TEXTLIST S6_Alarms
  0 = 'Station 6 Clamp A1 Failed to Advance... Check Q1.0...' | German: 'S6 0 Row 1 Failed To Advance.. Check Qxxx.x German' | French: 'S6 0 Row 1 Failed To Advance.. Check Qxxx.x French' | 汉语: '汉语'
  1 = 'Station 6 Clamp A1 Failed to Return... Check Q1.1...' | German: 'S6 1 Row 1 Failed To Return.. Check Qxxx.x German' | French: 'S6 1 Row 1 Failed To Return.. Check Qxxx.x French' | 汉语: '汉语'
  2 = 'Station 6 Clamp A1 Lost Advanced... Check I1.0...' | German: 'S6 2 Row 1 Lost Advance Position... Check Ixxx.x German' | French: 'S6 2 Row 1 Lost Advance Position... Check Ixxx.x French' | 汉语: '汉语'
  3 = 'Station 6 Clamp A1 Lost Returned... Check I1.1...' | German: 'S6 3 Row 1 Lost Return Position... Check Ixxx.x German' | French: 'S6 3 Row 1 Lost Return Position... Check Ixxx.x French' | 汉语: '汉语'
  4 = 'Station 6 Clamp A1 Switch Fault... Check I1.0, I1.1...' | German: 'S6 4 Row 1 Switch Fault... Check Ixxx.x / Ixxx.x German' | French: 'S6 4 Row 1 Switch Fault... Check Ixxx.x / Ixxx.x French'
  5 = 'Spare' | German: 'S6 5 Row 1 Spare Message German' | French: 'S6 5 Row 1 Spare Message French'
  6 = 'Spare' | German: 'S6 6 Row 1 Spare Message German' | French: 'S6 6 Row 1 Spare Message French'
  7 = 'Spare' | German: 'S6 7 Row 1 Spare Message German' | French: 'S6 7 Row 1 Spare Message French'
  8 = 'Spare' | German: 'S6 8 Row 1 Spare Message German' | French: 'S6 8 Row 1 Spare Message French'
  9 = 'Spare' | German: 'S6 9 Row 1 Spare Message German' | French: 'S6 9 Row 1 Spare Message French'
  10 = 'Lock Cylinder A2 Failed to Lock... Check Q1.2...' | German: 'S6 10 Row 2 Failed To Advance.. Check Qxxx.x German' | French: 'S6 10 Row 2 Failed To Advance.. Check Qxxx.x French'
  11 = 'Lock Cylinder A2 Failed to Unlock... Check Q1.3...' | German: 'S6 11 Row 2 Failed To Return.. Check Qxxx.x German' | French: 'S6 11 Row 2 Failed To Return.. Check Qxxx.x French'
  12 = 'Lock Cylinder A2 Lost Locked... Check I1.2...' | German: 'S6 12 Row 2 Lost Advance Position... Check Ixxx.x German' | French: 'S6 12 Row 2 Lost Advance Position... Check Ixxx.x French'
  13 = 'Lock Cylinder A2 Lost Unlocked... Check I1.3...' | German: 'S6 13 Row 2 Lost Return Position... Check Ixxx.x German' | French: 'S6 13 Row 2 Lost Return Position... Check Ixxx.x French'
  14 = 'Lock Cylinder A2 Switch Fault... Check I1.2, I1.3...' | German: 'S6 14 Row 2 Switch Fault... Check Ixxx.x / Ixxx.x German' | French: 'S6 14 Row 2 Switch Fault... Check Ixxx.x / Ixxx.x French'
  15 = 'Spare' | German: 'S6 15 Row 2 Spare Message German' | French: 'S6 15 Row 2 Spare Message French'
  16 = 'Spare' | German: 'S6 16 Row 2 Spare Message German' | French: 'S6 16 Row 2 Spare Message French'
  17 = 'Spare' | German: 'S6 17 Row 2 Spare Message German' | French: 'S6 17 Row 2 Spare Message French'
  18 = 'Spare' | German: 'S6 18 Row 2 Spare Message German' | French: 'S6 18 Row 2 Spare Message French'
  19 = 'Spare' | German: 'S6 19 Row 2 Spare Message German' | French: 'S6 19 Row 2 Spare Message French'
  20 = 'Urger Cylinder A3 Failed to Urge... Check Q1.4...' | German: 'S6 20 Row 3 Failed To Advance.. Check Qxxx.x German' | French: 'S6 20 Row 3 Failed To Advance.. Check Qxxx.x French'
  21 = 'Urger Cylinder A3 Failed to Return... Check Q1.5...' | German: 'S6 21 Row 3 Failed To Return.. Check Qxxx.x German' | French: 'S6 21 Row 3 Failed To Return.. Check Qxxx.x French'
  22 = 'Urger Cylinder A3 Lost Urged... Check I1.4...' | German: 'S6 22 Row 3 Lost Advance Position... Check Ixxx.x German' | French: 'S6 22 Row 3 Lost Advance Position... Check Ixxx.x French'
  23 = 'Urger Cylinder A3 Lost Returned... Check I1.5...' | German: 'S6 23 Row 3 Lost Return Position... Check Ixxx.x German' | French: 'S6 23 Row 3 Lost Return Position... Check Ixxx.x French'
  24 = 'Urger Cylinder A3 Switch Fault... Check I1.4, I1.5...' | German: 'S6 24 Row 3 Switch Fault... Check Ixxx.x / Ixxx.x German' | French: 'S6 24 Row 3 Switch Fault... Check Ixxx.x / Ixxx.x French'
  25 = 'Spare' | German: 'S6 25 Row 3 Spare Message German' | French: 'S6 25 Row 3 Spare Message French'
  26 = 'Spare' | German: 'S6 26 Row 3 Spare Message German' | French: 'S6 26 Row 3 Spare Message French'
  27 = 'Spare' | German: 'S6 27 Row 3 Spare Message German' | French: 'S6 27 Row 3 Spare Message French'
  28 = 'Spare' | German: 'S6 28 Row 3 Spare Message German' | French: 'S6 28 Row 3 Spare Message French'
  29 = 'Spare' | German: 'S6 29 Row 3 Spare Message German' | French: 'S6 29 Row 3 Spare Message French'
  30 = 'Clamp Cylinder A1 Failed to Advance... Check Q1.0...' | German: 'S6 30 Row 4 Failed To Advance.. Check Qxxx.x German' | French: 'S6 30 Row 4 Failed To Advance.. Check Qxxx.x French'
  31 = 'Clamp Cylinder A1 Failed to Return... Check Q1.1...' | German: 'S6 31 Row 4 Failed To Return.. Check Qxxx.x German' | French: 'S6 31 Row 4 Failed To Return.. Check Qxxx.x French'
  32 = 'Clamp Cylinder A1 Lost Advanced... Check I1.0...' | German: 'S6 32 Row 4 Lost Advance Position... Check Ixxx.x German' | French: 'S6 32 Row 4 Lost Advance Position... Check Ixxx.x French'
  33 = 'Clamp Cylinder A1 Lost Returned... Check I1.1...' | German: 'S6 33 Row 4 Lost Return Position... Check Ixxx.x German' | French: 'S6 33 Row 4 Lost Return Position... Check Ixxx.x French'
  34 = 'Clamp Cylinder A1 Switch Fault... Check I1.0, I1.1...' | German: 'S6 34 Row 4 Switch Fault... Check Ixxx.x / Ixxx.x German' | French: 'S6 34 Row 4 Switch Fault... Check Ixxx.x / Ixxx.x French'
  35 = 'Spare' | German: 'S6 35 Row 4 Spare Message German' | French: 'S6 35 Row 4 Spare Message French'
  36 = 'Spare' | German: 'S6 36 Row 4 Spare Message German' | French: 'S6 36 Row 4 Spare Message French'
  37 = 'Spare' | German: 'S6 37 Row 4 Spare Message German' | French: 'S6 37 Row 4 Spare Message French'
  38 = 'Spare' | German: 'S6 38 Row 4 Spare Message German' | French: 'S6 38 Row 4 Spare Message French'
  39 = 'Spare' | German: 'S6 39 Row 4 Spare Message German' | French: 'S6 39 Row 4 Spare Message French'
  40 = 'Clamp Cylinder A1 Failed to Advance... Check Q1.0...' | German: 'S6 40 Row 5 Failed To Advance.. Check Qxxx.x German' | French: 'S6 40 Row 5 Failed To Advance.. Check Qxxx.x French'
  41 = 'Clamp Cylinder A1 Failed to Return... Check Q1.1...' | German: 'S6 41 Row 5 Failed To Return.. Check Qxxx.x German' | French: 'S6 41 Row 5 Failed To Return.. Check Qxxx.x French'
  42 = 'Clamp Cylinder A1 Lost Advanced... Check I1.0...' | German: 'S6 42 Row 5 Lost Advance Position... Check Ixxx.x German' | French: 'S6 42 Row 5 Lost Advance Position... Check Ixxx.x French'
  43 = 'Clamp Cylinder A1 Lost Returned... Check I1.1...' | German: 'S6 43 Row 5 Lost Return Position... Check Ixxx.x German' | French: 'S6 43 Row 5 Lost Return Position... Check Ixxx.x French'
  44 = 'Clamp Cylinder A1 Switch Fault... Check I1.0, I1.1...' | German: 'S6 44 Row 5 Switch Fault... Check Ixxx.x / Ixxx.x German' | French: 'S6 44 Row 5 Switch Fault... Check Ixxx.x / Ixxx.x French'
  45 = 'Spare' | German: 'S6 45 Row 5 Spare Message German' | French: 'S6 45 Row 5 Spare Message French'
  46 = 'Spare' | German: 'S6 46 Row 5 Spare Message German' | French: 'S6 46 Row 5 Spare Message French'
  47 = 'Spare' | German: 'S6 47 Row 5 Spare Message German' | French: 'S6 47 Row 5 Spare Message French'
  48 = 'Spare' | German: 'S6 48 Row 5 Spare Message German' | French: 'S6 48 Row 5 Spare Message French'
  49 = 'Spare' | German: 'S6 49 Row 5 Spare Message German' | French: 'S6 49 Row 5 Spare Message French'
  50 = 'Clamp Cylinder A1 Failed to Advance... Check Q1.0...' | German: 'S6 50 Row 6 Failed To Advance.. Check Qxxx.x German' | French: 'S6 50 Row 6 Failed To Advance.. Check Qxxx.x French'
  51 = 'Clamp Cylinder A1 Failed to Return... Check Q1.1...' | German: 'S6 51 Row 6 Failed To Return.. Check Qxxx.x German' | French: 'S6 51 Row 6 Failed To Return.. Check Qxxx.x French'
  52 = 'Clamp Cylinder A1 Lost Advanced... Check I1.0...' | German: 'S6 52 Row 6 Lost Advance Position... Check Ixxx.x German' | French: 'S6 52 Row 6 Lost Advance Position... Check Ixxx.x French'
  53 = 'Clamp Cylinder A1 Lost Returned... Check I1.1...' | German: 'S6 53 Row 6 Lost Return Position... Check Ixxx.x German' | French: 'S6 53 Row 6 Lost Return Position... Check Ixxx.x French'
  54 = 'Clamp Cylinder A1 Switch Fault... Check I1.0, I1.1...' | German: 'S6 54 Row 6 Switch Fault... Check Ixxx.x / Ixxx.x German' | French: 'S6 54 Row 6 Switch Fault... Check Ixxx.x / Ixxx.x French'
  55 = 'Spare' | German: 'S6 55 Row 6 Spare Message German' | French: 'S6 55 Row 6 Spare Message French'
  56 = 'Spare' | German: 'S6 56 Row 6 Spare Message German' | French: 'S6 56 Row 6 Spare Message French'
  57 = 'Spare' | German: 'S6 57 Row 6 Spare Message German' | French: 'S6 57 Row 6 Spare Message French'
  58 = 'Spare' | German: 'S6 58 Row 6 Spare Message German' | French: 'S6 58 Row 6 Spare Message French'
  59 = 'Spare' | German: 'S6 59 Row 6 Spare Message German' | French: 'S6 59 Row 6 Spare Message French'
  60 = 'Clamp Cylinder A1 Failed to Advance... Check Q1.0...' | German: 'S6 60 Row 7 Failed To Advance.. Check Qxxx.x German' | French: 'S6 60 Row 7 Failed To Advance.. Check Qxxx.x French'
  61 = 'Clamp Cylinder A1 Failed to Return... Check Q1.1...' | German: 'S6 61 Row 7 Failed To Return.. Check Qxxx.x German' | French: 'S6 61 Row 7 Failed To Return.. Check Qxxx.x French'
  62 = 'Clamp Cylinder A1 Lost Advanced... Check I1.0...' | German: 'S6 62 Row 7 Lost Advance Position... Check Ixxx.x German' | French: 'S6 62 Row 7 Lost Advance Position... Check Ixxx.x French'
  63 = 'Clamp Cylinder A1 Lost Returned... Check I1.1...' | German: 'S6 63 Row 7 Lost Return Position... Check Ixxx.x German' | French: 'S6 63 Row 7 Lost Return Position... Check Ixxx.x French'
  64 = 'Clamp Cylinder A1 Switch Fault... Check I1.0, I1.1...' | German: 'S6 64 Row 7 Switch Fault... Check Ixxx.x / Ixxx.x German' | French: 'S6 64 Row 7 Switch Fault... Check Ixxx.x / Ixxx.x French'
  65 = 'Spare' | German: 'S6 65 Row 7 Spare Message German' | French: 'S6 65 Row 7 Spare Message French'
  66 = 'Spare' | German: 'S6 66 Row 7 Spare Message German' | French: 'S6 66 Row 7 Spare Message French'
  67 = 'Spare' | German: 'S6 67 Row 7 Spare Message German' | French: 'S6 67 Row 7 Spare Message French'
  68 = 'Spare' | German: 'S6 68 Row 7 Spare Message German' | French: 'S6 68 Row 7 Spare Message French'
  69 = 'Spare' | German: 'S6 69 Row 7 Spare Message German' | French: 'S6 69 Row 7 Spare Message French'
  70 = 'Clamp Cylinder A1 Failed to Advance... Check Q1.0...' | German: 'S6 70 Row 8 Failed To Advance.. Check Qxxx.x German' | French: 'S6 70 Row 8 Failed To Advance.. Check Qxxx.x French'
  71 = 'Clamp Cylinder A1 Failed to Return... Check Q1.1...' | German: 'S6 71 Row 8 Failed To Return.. Check Qxxx.x German' | French: 'S6 71 Row 8 Failed To Return.. Check Qxxx.x French'
  72 = 'Clamp Cylinder A1 Lost Advanced... Check I1.0...' | German: 'S6 72 Row 8 Lost Advance Position... Check Ixxx.x German' | French: 'S6 72 Row 8 Lost Advance Position... Check Ixxx.x French'
  73 = 'Clamp Cylinder A1 Lost Returned... Check I1.1...' | German: 'S6 73 Row 8 Lost Return Position... Check Ixxx.x German' | French: 'S6 73 Row 8 Lost Return Position... Check Ixxx.x French'
  74 = 'Clamp Cylinder A1 Switch Fault... Check I1.0, I1.1...' | German: 'S6 74 Row 8 Switch Fault... Check Ixxx.x / Ixxx.x German' | French: 'S6 74 Row 8 Switch Fault... Check Ixxx.x / Ixxx.x French'
  75 = 'Spare' | German: 'S6 75 Row 8 Spare Message German' | French: 'S6 75 Row 8 Spare Message French'
  76 = 'Spare' | German: 'S6 76 Row 8 Spare Message German' | French: 'S6 76 Row 8 Spare Message French'
  77 = 'Spare' | German: 'S6 77 Row 8 Spare Message German' | French: 'S6 77 Row 8 Spare Message French'
  78 = 'Spare' | German: 'S6 78 Row 8 Spare Message German' | French: 'S6 78 Row 8 Spare Message French'
  79 = 'Spare' | German: 'S6 79 Row 8 Spare Message German' | French: 'S6 79 Row 8 Spare Message French'
  80 = 'Clamp Cylinder A1 Failed to Advance... Check Q1.0...' | German: 'S6 80 Row 9 Failed To Advance.. Check Qxxx.x German' | French: 'S6 80 Row 9 Failed To Advance.. Check Qxxx.x French'
  81 = 'Clamp Cylinder A1 Failed to Return... Check Q1.1...' | German: 'S6 81 Row 9 Failed To Return.. Check Qxxx.x German' | French: 'S6 81 Row 9 Failed To Return.. Check Qxxx.x French'
  82 = 'Clamp Cylinder A1 Lost Advanced... Check I1.0...' | German: 'S6 82 Row 9 Lost Advance Position... Check Ixxx.x German' | French: 'S6 82 Row 9 Lost Advance Position... Check Ixxx.x French'
  83 = 'Clamp Cylinder A1 Lost Returned... Check I1.1...' | German: 'S6 83 Row 9 Lost Return Position... Check Ixxx.x German' | French: 'S6 83 Row 9 Lost Return Position... Check Ixxx.x French'
  84 = 'Clamp Cylinder A1 Switch Fault... Check I1.0, I1.1...' | German: 'S6 84 Row 9 Switch Fault... Check Ixxx.x / Ixxx.x German' | French: 'S6 84 Row 9 Switch Fault... Check Ixxx.x / Ixxx.x French'
  85 = 'Spare' | German: 'S6 85 Row 9 Spare Message German' | French: 'S6 85 Row 9 Spare Message French'
  86 = 'Spare' | German: 'S6 86 Row 9 Spare Message German' | French: 'S6 86 Row 9 Spare Message French'
  87 = 'Spare' | German: 'S6 87 Row 9 Spare Message German' | French: 'S6 87 Row 9 Spare Message French'
  88 = 'Spare' | German: 'S6 88 Row 9 Spare Message German' | French: 'S6 88 Row 9 Spare Message French'
  89 = 'Spare' | German: 'S6 89 Row 9 Spare Message German' | French: 'S6 89 Row 9 Spare Message French'
  90 = 'Clamp Cylinder A1 Failed to Advance... Check Q1.0...' | German: 'S6 90 Row 10 Failed To Advance.. Check Qxxx.x German' | French: 'S6 90 Row 10 Failed To Advance.. Check Qxxx.x French'
  91 = 'Clamp Cylinder A1 Failed to Return... Check Q1.1...' | German: 'S6 91 Row 10 Failed To Return.. Check Qxxx.x German' | French: 'S6 91 Row 10 Failed To Return.. Check Qxxx.x French'
  92 = 'Clamp Cylinder A1 Lost Advanced... Check I1.0...' | German: 'S6 92 Row 10 Lost Advance Position... Check Ixxx.x German' | French: 'S6 92 Row 10 Lost Advance Position... Check Ixxx.x French'
  93 = 'Clamp Cylinder A1 Lost Returned... Check I1.1...' | German: 'S6 93 Row 10 Lost Return Position... Check Ixxx.x German' | French: 'S6 93 Row 10 Lost Return Position... Check Ixxx.x French'
  94 = 'Clamp Cylinder A1 Switch Fault... Check I1.0, I1.1...' | German: 'S6 94 Row 10 Switch Fault... Check Ixxx.x / Ixxx.x German' | French: 'S6 94 Row 10 Switch Fault... Check Ixxx.x / Ixxx.x French'
  95 = 'Spare' | German: 'S6 95 Row 10 Spare Message German' | French: 'S6 95 Row 10 Spare Message French'
  96 = 'Spare' | German: 'S6 96 Row 10 Spare Message German' | French: 'S6 96 Row 10 Spare Message French'
  97 = 'Spare' | German: 'S6 97 Row 10 Spare Message German' | French: 'S6 97 Row 10 Spare Message French'
  98 = 'Spare' | German: 'S6 98 Row 10 Spare Message German' | French: 'S6 98 Row 10 Spare Message French'
  99 = 'Spare' | German: 'S6 99 Row 10 Spare Message German' | French: 'S6 99 Row 10 Spare Message French'
  100 = 'Clamp Cylinder A1 Failed to Advance... Check Q1.0...' | German: 'S6 100 Row 11 Failed To Advance.. Check Qxxx.x German' | French: 'S6 100 Row 11 Failed To Advance.. Check Qxxx.x French'
  101 = 'Clamp Cylinder A1 Failed to Return... Check Q1.1...' | German: 'S6 101 Row 11 Failed To Return.. Check Qxxx.x German' | French: 'S6 101 Row 11 Failed To Return.. Check Qxxx.x French'
  102 = 'Clamp Cylinder A1 Lost Advanced... Check I1.0...' | German: 'S6 102 Row 11 Lost Advance Position... Check Ixxx.x German' | French: 'S6 102 Row 11 Lost Advance Position... Check Ixxx.x French'
  103 = 'Clamp Cylinder A1 Lost Returned... Check I1.1...' | German: 'S6 103 Row 11 Lost Return Position... Check Ixxx.x German' | French: 'S6 103 Row 11 Lost Return Position... Check Ixxx.x French'
  104 = 'Clamp Cylinder A1 Switch Fault... Check I1.0, I1.1...' | German: 'S6 104 Row 11 Switch Fault... Check Ixxx.x / Ixxx.x German' | French: 'S6 104 Row 11 Switch Fault... Check Ixxx.x / Ixxx.x French'
  105 = 'Spare' | German: 'S6 105 Row 11 Spare Message German' | French: 'S6 105 Row 11 Spare Message French'
  106 = 'Spare' | German: 'S6 106 Row 11 Spare Message German' | French: 'S6 106 Row 11 Spare Message French'
  107 = 'Spare' | German: 'S6 107 Row 11 Spare Message German' | French: 'S6 107 Row 11 Spare Message French'
  108 = 'Spare' | German: 'S6 108 Row 11 Spare Message German' | French: 'S6 108 Row 11 Spare Message French'
  109 = 'Spare' | German: 'S6 109 Row 11 Spare Message German' | French: 'S6 109 Row 11 Spare Message French'
  110 = 'Clamp Cylinder A1 Failed to Advance... Check Q1.0...' | German: 'S6 110 Row 12 Failed To Advance.. Check Qxxx.x German' | French: 'S6 110 Row 12 Failed To Advance.. Check Qxxx.x French'
  111 = 'Clamp Cylinder A1 Failed to Return... Check Q1.1...' | German: 'S6 111 Row 12 Failed To Return.. Check Qxxx.x German' | French: 'S6 111 Row 12 Failed To Return.. Check Qxxx.x French'
  112 = 'Clamp Cylinder A1 Lost Advanced... Check I1.0...' | German: 'S6 112 Row 12 Lost Advance Position... Check Ixxx.x German' | French: 'S6 112 Row 12 Lost Advance Position... Check Ixxx.x French'
  113 = 'Clamp Cylinder A1 Lost Returned... Check I1.1...' | German: 'S6 113 Row 12 Lost Return Position... Check Ixxx.x German' | French: 'S6 113 Row 12 Lost Return Position... Check Ixxx.x French'
  114 = 'Clamp Cylinder A1 Switch Fault... Check I1.0, I1.1...' | German: 'S6 114 Row 12 Switch Fault... Check Ixxx.x / Ixxx.x German' | French: 'S6 114 Row 12 Switch Fault... Check Ixxx.x / Ixxx.x French'
  115 = 'Spare' | German: 'S6 115 Row 12 Spare Message German' | French: 'S6 115 Row 12 Spare Message French'
  116 = 'Spare' | German: 'S6 116 Row 12 Spare Message German' | French: 'S6 116 Row 12 Spare Message French'
  117 = 'Spare' | German: 'S6 117 Row 12 Spare Message German' | French: 'S6 117 Row 12 Spare Message French'
  118 = 'Spare' | German: 'S6 118 Row 12 Spare Message German' | French: 'S6 118 Row 12 Spare Message French'
  119 = 'Spare' | German: 'S6 119 Row 12 Spare Message German' | French: 'S6 119 Row 12 Spare Message French'
  120 = 'Clamp Cylinder A1 Failed to Advance... Check Q1.0...' | German: 'S6 120 Row 13 Failed To Advance.. Check Qxxx.x German' | French: 'S6 120 Row 13 Failed To Advance.. Check Qxxx.x French'
  121 = 'Clamp Cylinder A1 Failed to Return... Check Q1.1...' | German: 'S6 121 Row 13 Failed To Return.. Check Qxxx.x German' | French: 'S6 121 Row 13 Failed To Return.. Check Qxxx.x French'
  122 = 'Clamp Cylinder A1 Lost Advanced... Check I1.0...' | German: 'S6 122 Row 13 Lost Advance Position... Check Ixxx.x German' | French: 'S6 122 Row 13 Lost Advance Position... Check Ixxx.x French'
  123 = 'Clamp Cylinder A1 Lost Returned... Check I1.1...' | German: 'S6 123 Row 13 Lost Return Position... Check Ixxx.x German' | French: 'S6 123 Row 13 Lost Return Position... Check Ixxx.x French'
  124 = 'Clamp Cylinder A1 Switch Fault... Check I1.0, I1.1...' | German: 'S6 124 Row 13 Switch Fault... Check Ixxx.x / Ixxx.x German' | French: 'S6 124 Row 13 Switch Fault... Check Ixxx.x / Ixxx.x French'
  125 = 'Spare' | German: 'S6 125 Row 13 Spare Message German' | French: 'S6 125 Row 13 Spare Message French'
  126 = 'Spare' | German: 'S6 126 Row 13 Spare Message German' | French: 'S6 126 Row 13 Spare Message French'
  127 = 'Spare' | German: 'S6 127 Row 13 Spare Message German' | French: 'S6 127 Row 13 Spare Message French'
  128 = 'Spare' | German: 'S6 128 Row 13 Spare Message German' | French: 'S6 128 Row 13 Spare Message French'
  129 = 'Spare' | German: 'S6 129 Row 13 Spare Message German' | French: 'S6 129 Row 13 Spare Message French'
  130 = 'Clamp Cylinder A1 Failed to Advance... Check Q1.0...' | German: 'S6 130 Row 14 Failed To Advance.. Check Qxxx.x German' | French: 'S6 130 Row 14 Failed To Advance.. Check Qxxx.x French'
  131 = 'Clamp Cylinder A1 Failed to Return... Check Q1.1...' | German: 'S6 131 Row 14 Failed To Return.. Check Qxxx.x German' | French: 'S6 131 Row 14 Failed To Return.. Check Qxxx.x French'
  132 = 'Clamp Cylinder A1 Lost Advanced... Check I1.0...' | German: 'S6 132 Row 14 Lost Advance Position... Check Ixxx.x German' | French: 'S6 132 Row 14 Lost Advance Position... Check Ixxx.x French'
  133 = 'Clamp Cylinder A1 Lost Returned... Check I1.1...' | German: 'S6 133 Row 14 Lost Return Position... Check Ixxx.x German' | French: 'S6 133 Row 14 Lost Return Position... Check Ixxx.x French'
  134 = 'Clamp Cylinder A1 Switch Fault... Check I1.0, I1.1...' | German: 'S6 134 Row 14 Switch Fault... Check Ixxx.x / Ixxx.x German' | French: 'S6 134 Row 14 Switch Fault... Check Ixxx.x / Ixxx.x French'
  135 = 'Spare' | German: 'S6 135 Row 14 Spare Message German' | French: 'S6 135 Row 14 Spare Message French'
  136 = 'Spare' | German: 'S6 136 Row 14 Spare Message German' | French: 'S6 136 Row 14 Spare Message French'
  137 = 'Spare' | German: 'S6 137 Row 14 Spare Message German' | French: 'S6 137 Row 14 Spare Message French'
  138 = 'Spare' | German: 'S6 138 Row 14 Spare Message German' | French: 'S6 138 Row 14 Spare Message French'
  139 = 'Spare' | German: 'S6 139 Row 14 Spare Message German' | French: 'S6 139 Row 14 Spare Message French'
  140 = 'Clamp Cylinder A1 Failed to Advance... Check Q1.0...' | German: 'S6 140 Row 15 Failed To Advance.. Check Qxxx.x German' | French: 'S6 140 Row 15 Failed To Advance.. Check Qxxx.x French'
  141 = 'Clamp Cylinder A1 Failed to Return... Check Q1.1...' | German: 'S6 141 Row 15 Failed To Return.. Check Qxxx.x German' | French: 'S6 141 Row 15 Failed To Return.. Check Qxxx.x French'
  142 = 'Clamp Cylinder A1 Lost Advanced... Check I1.0...' | German: 'S6 142 Row 15 Lost Advance Position... Check Ixxx.x German' | French: 'S6 142 Row 15 Lost Advance Position... Check Ixxx.x French'
  143 = 'Clamp Cylinder A1 Lost Returned... Check I1.1...' | German: 'S6 143 Row 15 Lost Return Position... Check Ixxx.x German' | French: 'S6 143 Row 15 Lost Return Position... Check Ixxx.x French'
  144 = 'Clamp Cylinder A1 Switch Fault... Check I1.0, I1.1...' | German: 'S6 144 Row 15 Switch Fault... Check Ixxx.x / Ixxx.x German' | French: 'S6 144 Row 15 Switch Fault... Check Ixxx.x / Ixxx.x French'
  145 = 'Spare' | German: 'S6 145 Row 15 Spare Message German' | French: 'S6 145 Row 15 Spare Message French'
  146 = 'Spare' | German: 'S6 146 Row 15 Spare Message German' | French: 'S6 146 Row 15 Spare Message French'
  147 = 'Spare' | German: 'S6 147 Row 15 Spare Message German' | French: 'S6 147 Row 15 Spare Message French'
  148 = 'Spare' | German: 'S6 148 Row 15 Spare Message German' | French: 'S6 148 Row 15 Spare Message French'
  149 = 'Spare' | German: 'S6 149 Row 15 Spare Message German' | French: 'S6 149 Row 15 Spare Message French'
  150 = 'Clamp Cylinder A1 Failed to Advance... Check Q1.0...' | German: 'S6 150 Row 16 Failed To Advance.. Check Qxxx.x German' | French: 'S6 150 Row 16 Failed To Advance.. Check Qxxx.x French'
  151 = 'Clamp Cylinder A1 Failed to Return... Check Q1.1...' | German: 'S6 151 Row 16 Failed To Return.. Check Qxxx.x German' | French: 'S6 151 Row 16 Failed To Return.. Check Qxxx.x French'
  152 = 'Clamp Cylinder A1 Lost Advanced... Check I1.0...' | German: 'S6 152 Row 16 Lost Advance Position... Check Ixxx.x German' | French: 'S6 152 Row 16 Lost Advance Position... Check Ixxx.x French'
  153 = 'Clamp Cylinder A1 Lost Returned... Check I1.1...' | German: 'S6 153 Row 16 Lost Return Position... Check Ixxx.x German' | French: 'S6 153 Row 16 Lost Return Position... Check Ixxx.x French'
  154 = 'Clamp Cylinder A1 Switch Fault... Check I1.0, I1.1...' | German: 'S6 154 Row 16 Switch Fault... Check Ixxx.x / Ixxx.x German' | French: 'S6 154 Row 16 Switch Fault... Check Ixxx.x / Ixxx.x French'
  155 = 'Spare' | German: 'S6 155 Row 16 Spare Message German' | French: 'S6 155 Row 16 Spare Message French'
  156 = 'Spare' | German: 'S6 156 Row 16 Spare Message German' | French: 'S6 156 Row 16 Spare Message French'
  157 = 'Spare' | German: 'S6 157 Row 16 Spare Message German' | French: 'S6 157 Row 16 Spare Message French'
  158 = 'Spare' | German: 'S6 158 Row 16 Spare Message German' | French: 'S6 158 Row 16 Spare Message French'
  159 = 'Spare' | German: 'S6 159 Row 16 Spare Message German' | French: 'S6 159 Row 16 Spare Message French'
  160 = 'Clamp Cylinder A1 Failed to Advance... Check Q1.0...' | German: 'S6 160 Row 17 Failed To Advance.. Check Qxxx.x German' | French: 'S6 160 Row 17 Failed To Advance.. Check Qxxx.x French'
  161 = 'Clamp Cylinder A1 Failed to Return... Check Q1.1...' | German: 'S6 161 Row 17 Failed To Return.. Check Qxxx.x German' | French: 'S6 161 Row 17 Failed To Return.. Check Qxxx.x French'
  162 = 'Clamp Cylinder A1 Lost Advanced... Check I1.0...' | German: 'S6 162 Row 17 Lost Advance Position... Check Ixxx.x German' | French: 'S6 162 Row 17 Lost Advance Position... Check Ixxx.x French'
  163 = 'Clamp Cylinder A1 Lost Returned... Check I1.1...' | German: 'S6 163 Row 17 Lost Return Position... Check Ixxx.x German' | French: 'S6 163 Row 17 Lost Return Position... Check Ixxx.x French'
  164 = 'Clamp Cylinder A1 Switch Fault... Check I1.0, I1.1...' | German: 'S6 164 Row 17 Switch Fault... Check Ixxx.x / Ixxx.x German' | French: 'S6 164 Row 17 Switch Fault... Check Ixxx.x / Ixxx.x French'
  165 = 'Spare' | German: 'S6 165 Row 17 Spare Message German' | French: 'S6 165 Row 17 Spare Message French'
  166 = 'Spare' | German: 'S6 166 Row 17 Spare Message German' | French: 'S6 166 Row 17 Spare Message French'
  167 = 'Spare' | German: 'S6 167 Row 17 Spare Message German' | French: 'S6 167 Row 17 Spare Message French'
  168 = 'Spare' | German: 'S6 168 Row 17 Spare Message German' | French: 'S6 168 Row 17 Spare Message French'
  169 = 'Spare' | German: 'S6 169 Row 17 Spare Message German' | French: 'S6 169 Row 17 Spare Message French'
  170 = 'Clamp Cylinder A1 Failed to Advance... Check Q1.0...' | German: 'S6 170 Row 18 Failed To Advance.. Check Qxxx.x German' | French: 'S6 170 Row 18 Failed To Advance.. Check Qxxx.x French'
  171 = 'Clamp Cylinder A1 Failed to Return... Check Q1.1...' | German: 'S6 171 Row 18 Failed To Return.. Check Qxxx.x German' | French: 'S6 171 Row 18 Failed To Return.. Check Qxxx.x French'
  172 = 'Clamp Cylinder A1 Lost Advanced... Check I1.0...' | German: 'S6 172 Row 18 Lost Advance Position... Check Ixxx.x German' | French: 'S6 172 Row 18 Lost Advance Position... Check Ixxx.x French'
  173 = 'Clamp Cylinder A1 Lost Returned... Check I1.1...' | German: 'S6 173 Row 18 Lost Return Position... Check Ixxx.x German' | French: 'S6 173 Row 18 Lost Return Position... Check Ixxx.x French'
  174 = 'Clamp Cylinder A1 Switch Fault... Check I1.0, I1.1...' | German: 'S6 174 Row 18 Switch Fault... Check Ixxx.x / Ixxx.x German' | French: 'S6 174 Row 18 Switch Fault... Check Ixxx.x / Ixxx.x French'
  175 = 'Spare' | German: 'S6 175 Row 18 Spare Message German' | French: 'S6 175 Row 18 Spare Message French'
  176 = 'Spare' | German: 'S6 176 Row 18 Spare Message German' | French: 'S6 176 Row 18 Spare Message French'
  177 = 'Spare' | German: 'S6 177 Row 18 Spare Message German' | French: 'S6 177 Row 18 Spare Message French'
  178 = 'Spare' | German: 'S6 178 Row 18 Spare Message German' | French: 'S6 178 Row 18 Spare Message French'
  179 = 'Spare' | German: 'S6 179 Row 18 Spare Message German' | French: 'S6 179 Row 18 Spare Message French'
  180 = 'Clamp Cylinder A1 Failed to Advance... Check Q1.0...' | German: 'S6 180 Row 19 Failed To Advance.. Check Qxxx.x German' | French: 'S6 180 Row 19 Failed To Advance.. Check Qxxx.x French'
  181 = 'Clamp Cylinder A1 Failed to Return... Check Q1.1...' | German: 'S6 181 Row 19 Failed To Return.. Check Qxxx.x German' | French: 'S6 181 Row 19 Failed To Return.. Check Qxxx.x French'
  182 = 'Clamp Cylinder A1 Lost Advanced... Check I1.0...' | German: 'S6 182 Row 19 Lost Advance Position... Check Ixxx.x German' | French: 'S6 182 Row 19 Lost Advance Position... Check Ixxx.x French'
  183 = 'Clamp Cylinder A1 Lost Returned... Check I1.1...' | German: 'S6 183 Row 19 Lost Return Position... Check Ixxx.x German' | French: 'S6 183 Row 19 Lost Return Position... Check Ixxx.x French'
  184 = 'Clamp Cylinder A1 Switch Fault... Check I1.0, I1.1...' | German: 'S6 184 Row 19 Switch Fault... Check Ixxx.x / Ixxx.x German' | French: 'S6 184 Row 19 Switch Fault... Check Ixxx.x / Ixxx.x French'
  185 = 'Spare' | German: 'S6 185 Row 19 Spare Message German' | French: 'S6 185 Row 19 Spare Message French'
  186 = 'Spare' | German: 'S6 186 Row 19 Spare Message German' | French: 'S6 186 Row 19 Spare Message French'
  187 = 'Spare' | German: 'S6 187 Row 19 Spare Message German' | French: 'S6 187 Row 19 Spare Message French'
  188 = 'Spare' | German: 'S6 188 Row 19 Spare Message German' | French: 'S6 188 Row 19 Spare Message French'
  189 = 'Spare' | German: 'S6 189 Row 19 Spare Message German' | French: 'S6 189 Row 19 Spare Message French'
  190 = 'Clamp Cylinder A1 Failed to Advance... Check Q1.0...' | German: 'S6 190 Row 20 Failed To Advance.. Check Qxxx.x German' | French: 'S6 190 Row 20 Failed To Advance.. Check Qxxx.x French'
  191 = 'Clamp Cylinder A1 Failed to Return... Check Q1.1...' | German: 'S6 191 Row 20 Failed To Return.. Check Qxxx.x German' | French: 'S6 191 Row 20 Failed To Return.. Check Qxxx.x French'
  192 = 'Clamp Cylinder A1 Lost Advanced... Check I1.0...' | German: 'S6 192 Row 20 Lost Advance Position... Check Ixxx.x German' | French: 'S6 192 Row 20 Lost Advance Position... Check Ixxx.x French'
  193 = 'Clamp Cylinder A1 Lost Returned... Check I1.1...' | German: 'S6 193 Row 20 Lost Return Position... Check Ixxx.x German' | French: 'S6 193 Row 20 Lost Return Position... Check Ixxx.x French'
  194 = 'Clamp Cylinder A1 Switch Fault... Check I1.0, I1.1...' | German: 'S6 194 Row 20 Switch Fault... Check Ixxx.x / Ixxx.x German' | French: 'S6 194 Row 20 Switch Fault... Check Ixxx.x / Ixxx.x French'
  195 = 'Spare' | German: 'S6 195 Row 20 Spare Message German' | French: 'S6 195 Row 20 Spare Message French'
  196 = 'Spare' | German: 'S6 196 Row 20 Spare Message German' | French: 'S6 196 Row 20 Spare Message French'
  197 = 'Spare' | German: 'S6 197 Row 20 Spare Message German' | French: 'S6 197 Row 20 Spare Message French'
  198 = 'Spare' | German: 'S6 198 Row 20 Spare Message German' | French: 'S6 198 Row 20 Spare Message French'
  199 = 'Spare' | German: 'S6 199 Row 20 Spare Message German' | French: 'S6 199 Row 20 Spare Message French'
  200 = 'Clamp Cylinder A1 Failed to Advance... Check Q1.0...' | German: 'S6 200 Row 21 Failed To Advance.. Check Qxxx.x German' | French: 'S6 200 Row 21 Failed To Advance.. Check Qxxx.x French'
  201 = 'Clamp Cylinder A1 Failed to Return... Check Q1.1...' | German: 'S6 201 Row 21 Failed To Return.. Check Qxxx.x German' | French: 'S6 201 Row 21 Failed To Return.. Check Qxxx.x French'
  202 = 'Clamp Cylinder A1 Lost Advanced... Check I1.0...' | German: 'S6 202 Row 21 Lost Advance Position... Check Ixxx.x German' | French: 'S6 202 Row 21 Lost Advance Position... Check Ixxx.x French'
  203 = 'Clamp Cylinder A1 Lost Returned... Check I1.1...' | German: 'S6 203 Row 21 Lost Return Position... Check Ixxx.x German' | French: 'S6 203 Row 21 Lost Return Position... Check Ixxx.x French'
  204 = 'Clamp Cylinder A1 Switch Fault... Check I1.0, I1.1...' | German: 'S6 204 Row 21 Switch Fault... Check Ixxx.x / Ixxx.x German' | French: 'S6 204 Row 21 Switch Fault... Check Ixxx.x / Ixxx.x French'
  205 = 'Spare' | German: 'S6 205 Row 21 Spare Message German' | French: 'S6 205 Row 21 Spare Message French'
  206 = 'Spare' | German: 'S6 206 Row 21 Spare Message German' | French: 'S6 206 Row 21 Spare Message French'
  207 = 'Spare' | German: 'S6 207 Row 21 Spare Message German' | French: 'S6 207 Row 21 Spare Message French'
  208 = 'Spare' | German: 'S6 208 Row 21 Spare Message German' | French: 'S6 208 Row 21 Spare Message French'
  209 = 'Spare' | German: 'S6 209 Row 21 Spare Message German' | French: 'S6 209 Row 21 Spare Message French'
  210 = 'Clamp Cylinder A1 Failed to Advance... Check Q1.0...' | German: 'S6 210 Row 22 Failed To Advance.. Check Qxxx.x German' | French: 'S6 210 Row 22 Failed To Advance.. Check Qxxx.x French'
  211 = 'Clamp Cylinder A1 Failed to Return... Check Q1.1...' | German: 'S6 211 Row 22 Failed To Return.. Check Qxxx.x German' | French: 'S6 211 Row 22 Failed To Return.. Check Qxxx.x French'
  212 = 'Clamp Cylinder A1 Lost Advanced... Check I1.0...' | German: 'S6 212 Row 22 Lost Advance Position... Check Ixxx.x German' | French: 'S6 212 Row 22 Lost Advance Position... Check Ixxx.x French'
  213 = 'Clamp Cylinder A1 Lost Returned... Check I1.1...' | German: 'S6 213 Row 22 Lost Return Position... Check Ixxx.x German' | French: 'S6 213 Row 22 Lost Return Position... Check Ixxx.x French'
  214 = 'Clamp Cylinder A1 Switch Fault... Check I1.0, I1.1...' | German: 'S6 214 Row 22 Switch Fault... Check Ixxx.x / Ixxx.x German' | French: 'S6 214 Row 22 Switch Fault... Check Ixxx.x / Ixxx.x French'
  215 = 'Spare' | German: 'S6 215 Row 22 Spare Message German' | French: 'S6 215 Row 22 Spare Message French'
  216 = 'Spare' | German: 'S6 216 Row 22 Spare Message German' | French: 'S6 216 Row 22 Spare Message French'
  217 = 'Spare' | German: 'S6 217 Row 22 Spare Message German' | French: 'S6 217 Row 22 Spare Message French'
  218 = 'Spare' | German: 'S6 218 Row 22 Spare Message German' | French: 'S6 218 Row 22 Spare Message French'
  219 = 'Spare' | German: 'S6 219 Row 22 Spare Message German' | French: 'S6 219 Row 22 Spare Message French'
  220 = 'Clamp Cylinder A1 Failed to Advance... Check Q1.0...' | German: 'S6 220 Row 23 Failed To Advance.. Check Qxxx.x German' | French: 'S6 220 Row 23 Failed To Advance.. Check Qxxx.x French'
  221 = 'Clamp Cylinder A1 Failed to Return... Check Q1.1...' | German: 'S6 221 Row 23 Failed To Return.. Check Qxxx.x German' | French: 'S6 221 Row 23 Failed To Return.. Check Qxxx.x French'
  222 = 'Clamp Cylinder A1 Lost Advanced... Check I1.0...' | German: 'S6 222 Row 23 Lost Advance Position... Check Ixxx.x German' | French: 'S6 222 Row 23 Lost Advance Position... Check Ixxx.x French'
  223 = 'Clamp Cylinder A1 Lost Returned... Check I1.1...' | German: 'S6 223 Row 23 Lost Return Position... Check Ixxx.x German' | French: 'S6 223 Row 23 Lost Return Position... Check Ixxx.x French'
  224 = 'Clamp Cylinder A1 Switch Fault... Check I1.0, I1.1...' | German: 'S6 224 Row 23 Switch Fault... Check Ixxx.x / Ixxx.x German' | French: 'S6 224 Row 23 Switch Fault... Check Ixxx.x / Ixxx.x French'
  225 = 'Spare' | German: 'S6 225 Row 23 Spare Message German' | French: 'S6 225 Row 23 Spare Message French'
  226 = 'Spare' | German: 'S6 226 Row 23 Spare Message German' | French: 'S6 226 Row 23 Spare Message French'
  227 = 'Spare' | German: 'S6 227 Row 23 Spare Message German' | French: 'S6 227 Row 23 Spare Message French'
  228 = 'Spare' | German: 'S6 228 Row 23 Spare Message German' | French: 'S6 228 Row 23 Spare Message French'
  229 = 'Spare' | German: 'S6 229 Row 23 Spare Message German' | French: 'S6 229 Row 23 Spare Message French'
  230 = 'Clamp Cylinder A1 Failed to Advance... Check Q1.0...' | German: 'S6 230 Row 24 Failed To Advance.. Check Qxxx.x German' | French: 'S6 230 Row 24 Failed To Advance.. Check Qxxx.x French'
  231 = 'Clamp Cylinder A1 Failed to Return... Check Q1.1...' | German: 'S6 231 Row 24 Failed To Return.. Check Qxxx.x German' | French: 'S6 231 Row 24 Failed To Return.. Check Qxxx.x French'
  232 = 'Clamp Cylinder A1 Lost Advanced... Check I1.0...' | German: 'S6 232 Row 24 Lost Advance Position... Check Ixxx.x German' | French: 'S6 232 Row 24 Lost Advance Position... Check Ixxx.x French'
  233 = 'Clamp Cylinder A1 Lost Returned... Check I1.1...' | German: 'S6 233 Row 24 Lost Return Position... Check Ixxx.x German' | French: 'S6 233 Row 24 Lost Return Position... Check Ixxx.x French'
  234 = 'Clamp Cylinder A1 Switch Fault... Check I1.0, I1.1...' | German: 'S6 234 Row 24 Switch Fault... Check Ixxx.x / Ixxx.x German' | French: 'S6 234 Row 24 Switch Fault... Check Ixxx.x / Ixxx.x French'
  235 = 'Spare' | German: 'S6 235 Row 24 Spare Message German' | French: 'S6 235 Row 24 Spare Message French'
  236 = 'Spare' | German: 'S6 236 Row 24 Spare Message German' | French: 'S6 236 Row 24 Spare Message French'
  237 = 'Spare' | German: 'S6 237 Row 24 Spare Message German' | French: 'S6 237 Row 24 Spare Message French'
  238 = 'Spare' | German: 'S6 238 Row 24 Spare Message German' | French: 'S6 238 Row 24 Spare Message French'
  239 = 'Spare' | German: 'S6 239 Row 24 Spare Message German' | French: 'S6 239 Row 24 Spare Message French'
  240 = 'Clamp Cylinder A1 Failed to Advance... Check Q1.0...' | German: 'S6 240 Row 25 Failed To Advance.. Check Qxxx.x German' | French: 'S6 240 Row 25 Failed To Advance.. Check Qxxx.x French'
  241 = 'Clamp Cylinder A1 Failed to Return... Check Q1.1...' | German: 'S6 241 Row 25 Failed To Return.. Check Qxxx.x German' | French: 'S6 241 Row 25 Failed To Return.. Check Qxxx.x French'
  242 = 'Clamp Cylinder A1 Lost Advanced... Check I1.0...' | German: 'S6 242 Row 25 Lost Advance Position... Check Ixxx.x German' | French: 'S6 242 Row 25 Lost Advance Position... Check Ixxx.x French'
  243 = 'Clamp Cylinder A1 Lost Returned... Check I1.1...' | German: 'S6 243 Row 25 Lost Return Position... Check Ixxx.x German' | French: 'S6 243 Row 25 Lost Return Position... Check Ixxx.x French'
  244 = 'Clamp Cylinder A1 Switch Fault... Check I1.0, I1.1...' | German: 'S6 244 Row 25 Switch Fault... Check Ixxx.x / Ixxx.x German' | French: 'S6 244 Row 25 Switch Fault... Check Ixxx.x / Ixxx.x French'
  245 = 'Spare' | German: 'S6 245 Row 25 Spare Message German' | French: 'S6 245 Row 25 Spare Message French'
  246 = 'Spare' | German: 'S6 246 Row 25 Spare Message German' | French: 'S6 246 Row 25 Spare Message French'
  247 = 'Spare' | German: 'S6 247 Row 25 Spare Message German' | French: 'S6 247 Row 25 Spare Message French'
  248 = 'Spare' | German: 'S6 248 Row 25 Spare Message German' | French: 'S6 248 Row 25 Spare Message French'
  249 = 'Spare' | German: 'S6 249 Row 25 Spare Message German' | French: 'S6 249 Row 25 Spare Message French'
  250 = 'Clamp Cylinder A1 Failed to Advance... Check Q1.0...' | German: 'S6 250 Row 26 Failed To Advance.. Check Qxxx.x German' | French: 'S6 250 Row 26 Failed To Advance.. Check Qxxx.x French'
  251 = 'Clamp Cylinder A1 Failed to Return... Check Q1.1...' | German: 'S6 251 Row 26 Failed To Return.. Check Qxxx.x German' | French: 'S6 251 Row 26 Failed To Return.. Check Qxxx.x French'
  252 = 'Clamp Cylinder A1 Lost Advanced... Check I1.0...' | German: 'S6 252 Row 26 Lost Advance Position... Check Ixxx.x German' | French: 'S6 252 Row 26 Lost Advance Position... Check Ixxx.x French'
  253 = 'Clamp Cylinder A1 Lost Returned... Check I1.1...' | German: 'S6 253 Row 26 Lost Return Position... Check Ixxx.x German' | French: 'S6 253 Row 26 Lost Return Position... Check Ixxx.x French'
  254 = 'Clamp Cylinder A1 Switch Fault... Check I1.0, I1.1...' | German: 'S6 254 Row 26 Switch Fault... Check Ixxx.x / Ixxx.x German' | French: 'S6 254 Row 26 Switch Fault... Check Ixxx.x / Ixxx.x French'
  255 = 'Spare' | German: 'S6 255 Row 26 Spare Message German' | French: 'S6 255 Row 26 Spare Message French'
  256 = 'Spare' | German: 'S6 256 Row 26 Spare Message German' | French: 'S6 256 Row 26 Spare Message French'
  257 = 'Spare' | German: 'S6 257 Row 26 Spare Message German' | French: 'S6 257 Row 26 Spare Message French'
  258 = 'Spare' | German: 'S6 258 Row 26 Spare Message German' | French: 'S6 258 Row 26 Spare Message French'
  259 = 'Spare' | German: 'S6 259 Row 26 Spare Message German' | French: 'S6 259 Row 26 Spare Message French'
  260 = 'Clamp Cylinder A1 Failed to Advance... Check Q1.0...' | German: 'S6 260 Row 27 Failed To Advance.. Check Qxxx.x German' | French: 'S6 260 Row 27 Failed To Advance.. Check Qxxx.x French'
  261 = 'Clamp Cylinder A1 Failed to Return... Check Q1.1...' | German: 'S6 261 Row 27 Failed To Return.. Check Qxxx.x German' | French: 'S6 261 Row 27 Failed To Return.. Check Qxxx.x French'
  262 = 'Clamp Cylinder A1 Lost Advanced... Check I1.0...' | German: 'S6 262 Row 27 Lost Advance Position... Check Ixxx.x German' | French: 'S6 262 Row 27 Lost Advance Position... Check Ixxx.x French'
  263 = 'Clamp Cylinder A1 Lost Returned... Check I1.1...' | German: 'S6 263 Row 27 Lost Return Position... Check Ixxx.x German' | French: 'S6 263 Row 27 Lost Return Position... Check Ixxx.x French'
  264 = 'Clamp Cylinder A1 Switch Fault... Check I1.0, I1.1...' | German: 'S6 264 Row 27 Switch Fault... Check Ixxx.x / Ixxx.x German' | French: 'S6 264 Row 27 Switch Fault... Check Ixxx.x / Ixxx.x French'
  265 = 'Spare' | German: 'S6 265 Row 27 Spare Message German' | French: 'S6 265 Row 27 Spare Message French'
  266 = 'Spare' | German: 'S6 266 Row 27 Spare Message German' | French: 'S6 266 Row 27 Spare Message French'
  267 = 'Spare' | German: 'S6 267 Row 27 Spare Message German' | French: 'S6 267 Row 27 Spare Message French'
  268 = 'Spare' | German: 'S6 268 Row 27 Spare Message German' | French: 'S6 268 Row 27 Spare Message French'
  269 = 'Spare' | German: 'S6 269 Row 27 Spare Message German' | French: 'S6 269 Row 27 Spare Message French'
  270 = 'Clamp Cylinder A1 Failed to Advance... Check Q1.0...' | German: 'S6 270 Row 28 Failed To Advance.. Check Qxxx.x German' | French: 'S6 270 Row 28 Failed To Advance.. Check Qxxx.x French'
  271 = 'Clamp Cylinder A1 Failed to Return... Check Q1.1...' | German: 'S6 271 Row 28 Failed To Return.. Check Qxxx.x German' | French: 'S6 271 Row 28 Failed To Return.. Check Qxxx.x French'
  272 = 'Clamp Cylinder A1 Lost Advanced... Check I1.0...' | German: 'S6 272 Row 28 Lost Advance Position... Check Ixxx.x German' | French: 'S6 272 Row 28 Lost Advance Position... Check Ixxx.x French'
  273 = 'Clamp Cylinder A1 Lost Returned... Check I1.1...' | German: 'S6 273 Row 28 Lost Return Position... Check Ixxx.x German' | French: 'S6 273 Row 28 Lost Return Position... Check Ixxx.x French'
  274 = 'Clamp Cylinder A1 Switch Fault... Check I1.0, I1.1...' | German: 'S6 274 Row 28 Switch Fault... Check Ixxx.x / Ixxx.x German' | French: 'S6 274 Row 28 Switch Fault... Check Ixxx.x / Ixxx.x French'
  275 = 'Spare' | German: 'S6 275 Row 28 Spare Message German' | French: 'S6 275 Row 28 Spare Message French'
  276 = 'Spare' | German: 'S6 276 Row 28 Spare Message German' | French: 'S6 276 Row 28 Spare Message French'
  277 = 'Spare' | German: 'S6 277 Row 28 Spare Message German' | French: 'S6 277 Row 28 Spare Message French'
  278 = 'Spare' | German: 'S6 278 Row 28 Spare Message German' | French: 'S6 278 Row 28 Spare Message French'
  279 = 'Spare' | German: 'S6 279 Row 28 Spare Message German' | French: 'S6 279 Row 28 Spare Message French'
  280 = 'Clamp Cylinder A1 Failed to Advance... Check Q1.0...' | German: 'S6 280 Row 29 Failed To Advance.. Check Qxxx.x German' | French: 'S6 280 Row 29 Failed To Advance.. Check Qxxx.x French'
  281 = 'Clamp Cylinder A1 Failed to Return... Check Q1.1...' | German: 'S6 281 Row 29 Failed To Return.. Check Qxxx.x German' | French: 'S6 281 Row 29 Failed To Return.. Check Qxxx.x French'
  282 = 'Clamp Cylinder A1 Lost Advanced... Check I1.0...' | German: 'S6 282 Row 29 Lost Advance Position... Check Ixxx.x German' | French: 'S6 282 Row 29 Lost Advance Position... Check Ixxx.x French'
  283 = 'Clamp Cylinder A1 Lost Returned... Check I1.1...' | German: 'S6 283 Row 29 Lost Return Position... Check Ixxx.x German' | French: 'S6 283 Row 29 Lost Return Position... Check Ixxx.x French'
  284 = 'Clamp Cylinder A1 Switch Fault... Check I1.0, I1.1...' | German: 'S6 284 Row 29 Switch Fault... Check Ixxx.x / Ixxx.x German' | French: 'S6 284 Row 29 Switch Fault... Check Ixxx.x / Ixxx.x French'
  285 = 'Spare' | German: 'S6 285 Row 29 Spare Message German' | French: 'S6 285 Row 29 Spare Message French'
  286 = 'Spare' | German: 'S6 286 Row 29 Spare Message German' | French: 'S6 286 Row 29 Spare Message French'
  287 = 'Spare' | German: 'S6 287 Row 29 Spare Message German' | French: 'S6 287 Row 29 Spare Message French'
  288 = 'Spare' | German: 'S6 288 Row 29 Spare Message German' | French: 'S6 288 Row 29 Spare Message French'
  289 = 'Spare' | German: 'S6 289 Row 29 Spare Message German' | French: 'S6 289 Row 29 Spare Message French'
  290 = 'Clamp Cylinder A1 Failed to Advance... Check Q1.0...' | German: 'S6 290 Row 30 Failed To Advance.. Check Qxxx.x German' | French: 'S6 290 Row 30 Failed To Advance.. Check Qxxx.x French'
  291 = 'Clamp Cylinder A1 Failed to Return... Check Q1.1...' | German: 'S6 291 Row 30 Failed To Return.. Check Qxxx.x German' | French: 'S6 291 Row 30 Failed To Return.. Check Qxxx.x French'
  292 = 'Clamp Cylinder A1 Lost Advanced... Check I1.0...' | German: 'S6 292 Row 30 Lost Advance Position... Check Ixxx.x German' | French: 'S6 292 Row 30 Lost Advance Position... Check Ixxx.x French'
  293 = 'Clamp Cylinder A1 Lost Returned... Check I1.1...' | German: 'S6 293 Row 30 Lost Return Position... Check Ixxx.x German' | French: 'S6 293 Row 30 Lost Return Position... Check Ixxx.x French'
  294 = 'Clamp Cylinder A1 Switch Fault... Check I1.0, I1.1...' | German: 'S6 294 Row 30 Switch Fault... Check Ixxx.x / Ixxx.x German' | French: 'S6 294 Row 30 Switch Fault... Check Ixxx.x / Ixxx.x French'
  295 = 'Spare' | German: 'S6 295 Row 30 Spare Message German' | French: 'S6 295 Row 30 Spare Message French'
  296 = 'Spare' | German: 'S6 296 Row 30 Spare Message German' | French: 'S6 296 Row 30 Spare Message French'
  297 = 'Spare' | German: 'S6 297 Row 30 Spare Message German' | French: 'S6 297 Row 30 Spare Message French'
  298 = 'Spare' | German: 'S6 298 Row 30 Spare Message German' | French: 'S6 298 Row 30 Spare Message French'
  299 = 'Spare' | German: 'S6 299 Row 30 Spare Message German' | French: 'S6 299 Row 30 Spare Message French'
  300 = 'Clamp Cylinder A1 Failed to Advance... Check Q1.0...' | German: 'S6 300 Row 31 Failed To Advance.. Check Qxxx.x German' | French: 'S6 300 Row 31 Failed To Advance.. Check Qxxx.x French'
  301 = 'Clamp Cylinder A1 Failed to Return... Check Q1.1...' | German: 'S6 301 Row 31 Failed To Return.. Check Qxxx.x German' | French: 'S6 301 Row 31 Failed To Return.. Check Qxxx.x French'
  302 = 'Clamp Cylinder A1 Lost Advanced... Check I1.0...' | German: 'S6 302 Row 31 Lost Advance Position... Check Ixxx.x German' | French: 'S6 302 Row 31 Lost Advance Position... Check Ixxx.x French'
  303 = 'Clamp Cylinder A1 Lost Returned... Check I1.1...' | German: 'S6 303 Row 31 Lost Return Position... Check Ixxx.x German' | French: 'S6 303 Row 31 Lost Return Position... Check Ixxx.x French'
  304 = 'Clamp Cylinder A1 Switch Fault... Check I1.0, I1.1...' | German: 'S6 304 Row 31 Switch Fault... Check Ixxx.x / Ixxx.x German' | French: 'S6 304 Row 31 Switch Fault... Check Ixxx.x / Ixxx.x French'
  305 = 'Spare' | German: 'S6 305 Row 31 Spare Message German' | French: 'S6 305 Row 31 Spare Message French'
  306 = 'Spare' | German: 'S6 306 Row 31 Spare Message German' | French: 'S6 306 Row 31 Spare Message French'
  307 = 'Spare' | German: 'S6 307 Row 31 Spare Message German' | French: 'S6 307 Row 31 Spare Message French'
  308 = 'Spare' | German: 'S6 308 Row 31 Spare Message German' | French: 'S6 308 Row 31 Spare Message French'
  309 = 'Spare' | German: 'S6 309 Row 31 Spare Message German' | French: 'S6 309 Row 31 Spare Message French'
  310 = 'Clamp Cylinder A1 Failed to Advance... Check Q1.0...' | German: 'S6 310 Row 32 Failed To Advance.. Check Qxxx.x German' | French: 'S6 310 Row 32 Failed To Advance.. Check Qxxx.x French'
  311 = 'Clamp Cylinder A1 Failed to Return... Check Q1.1...' | German: 'S6 311 Row 32 Failed To Return.. Check Qxxx.x German' | French: 'S6 311 Row 32 Failed To Return.. Check Qxxx.x French'
  312 = 'Clamp Cylinder A1 Lost Advanced... Check I1.0...' | German: 'S6 312 Row 32 Lost Advance Position... Check Ixxx.x German' | French: 'S6 312 Row 32 Lost Advance Position... Check Ixxx.x French'
  313 = 'Clamp Cylinder A1 Lost Returned... Check I1.1...' | German: 'S6 313 Row 32 Lost Return Position... Check Ixxx.x German' | French: 'S6 313 Row 32 Lost Return Position... Check Ixxx.x French'
  314 = 'Clamp Cylinder A1 Switch Fault... Check I1.0, I1.1...' | German: 'S6 314 Row 32 Switch Fault... Check Ixxx.x / Ixxx.x German' | French: 'S6 314 Row 32 Switch Fault... Check Ixxx.x / Ixxx.x French'
  315 = 'Spare' | German: 'S6 315 Row 32 Spare Message German' | French: 'S6 315 Row 32 Spare Message French'
  316 = 'Spare' | German: 'S6 316 Row 32 Spare Message German' | French: 'S6 316 Row 32 Spare Message French'
  317 = 'Spare' | German: 'S6 317 Row 32 Spare Message German' | French: 'S6 317 Row 32 Spare Message French'
  318 = 'Spare' | German: 'S6 318 Row 32 Spare Message German' | French: 'S6 318 Row 32 Spare Message French'
  319 = 'Spare' | German: 'S6 319 Row 32 Spare Message German' | French: 'S6 319 Row 32 Spare Message French'
  320 = 'Clamp Cylinder A1 Failed to Advance... Check Q1.0...' | German: 'S6 320 Row 33 Failed To Advance.. Check Qxxx.x German' | French: 'S6 320 Row 33 Failed To Advance.. Check Qxxx.x French'
  321 = 'Clamp Cylinder A1 Failed to Return... Check Q1.1...' | German: 'S6 321 Row 33 Failed To Return.. Check Qxxx.x German' | French: 'S6 321 Row 33 Failed To Return.. Check Qxxx.x French'
  322 = 'Clamp Cylinder A1 Lost Advanced... Check I1.0...' | German: 'S6 322 Row 33 Lost Advance Position... Check Ixxx.x German' | French: 'S6 322 Row 33 Lost Advance Position... Check Ixxx.x French'
  323 = 'Clamp Cylinder A1 Lost Returned... Check I1.1...' | German: 'S6 323 Row 33 Lost Return Position... Check Ixxx.x German' | French: 'S6 323 Row 33 Lost Return Position... Check Ixxx.x French'
  324 = 'Clamp Cylinder A1 Switch Fault... Check I1.0, I1.1...' | German: 'S6 324 Row 33 Switch Fault... Check Ixxx.x / Ixxx.x German' | French: 'S6 324 Row 33 Switch Fault... Check Ixxx.x / Ixxx.x French'
  325 = 'Spare' | German: 'S6 325 Row 33 Spare Message German' | French: 'S6 325 Row 33 Spare Message French'
  326 = 'Spare' | German: 'S6 326 Row 33 Spare Message German' | French: 'S6 326 Row 33 Spare Message French'
  327 = 'Spare' | German: 'S6 327 Row 33 Spare Message German' | French: 'S6 327 Row 33 Spare Message French'
  328 = 'Spare' | German: 'S6 328 Row 33 Spare Message German' | French: 'S6 328 Row 33 Spare Message French'
  329 = 'Spare' | German: 'S6 329 Row 33 Spare Message German' | French: 'S6 329 Row 33 Spare Message French'
  330 = 'Clamp Cylinder A1 Failed to Advance... Check Q1.0...' | German: 'S6 330 Row 34 Failed To Advance.. Check Qxxx.x German' | French: 'S6 330 Row 34 Failed To Advance.. Check Qxxx.x French'
  331 = 'Clamp Cylinder A1 Failed to Return... Check Q1.1...' | German: 'S6 331 Row 34 Failed To Return.. Check Qxxx.x German' | French: 'S6 331 Row 34 Failed To Return.. Check Qxxx.x French'
  332 = 'Clamp Cylinder A1 Lost Advanced... Check I1.0...' | German: 'S6 332 Row 34 Lost Advance Position... Check Ixxx.x German' | French: 'S6 332 Row 34 Lost Advance Position... Check Ixxx.x French'
  333 = 'Clamp Cylinder A1 Lost Returned... Check I1.1...' | German: 'S6 333 Row 34 Lost Return Position... Check Ixxx.x German' | French: 'S6 333 Row 34 Lost Return Position... Check Ixxx.x French'
  334 = 'Clamp Cylinder A1 Switch Fault... Check I1.0, I1.1...' | German: 'S6 334 Row 34 Switch Fault... Check Ixxx.x / Ixxx.x German' | French: 'S6 334 Row 34 Switch Fault... Check Ixxx.x / Ixxx.x French'
  335 = 'Spare' | German: 'S6 335 Row 34 Spare Message German' | French: 'S6 335 Row 34 Spare Message French'
  336 = 'Spare' | German: 'S6 336 Row 34 Spare Message German' | French: 'S6 336 Row 34 Spare Message French'
  337 = 'Spare' | German: 'S6 337 Row 34 Spare Message German' | French: 'S6 337 Row 34 Spare Message French'
  338 = 'Spare' | German: 'S6 338 Row 34 Spare Message German' | French: 'S6 338 Row 34 Spare Message French'
  339 = 'Spare' | German: 'S6 339 Row 34 Spare Message German' | French: 'S6 339 Row 34 Spare Message French'
  340 = 'Clamp Cylinder A1 Failed to Advance... Check Q1.0...' | German: 'S6 340 Row 35 Failed To Advance.. Check Qxxx.x German' | French: 'S6 340 Row 35 Failed To Advance.. Check Qxxx.x French'
  341 = 'Clamp Cylinder A1 Failed to Return... Check Q1.1...' | German: 'S6 341 Row 35 Failed To Return.. Check Qxxx.x German' | French: 'S6 341 Row 35 Failed To Return.. Check Qxxx.x French'
  342 = 'Clamp Cylinder A1 Lost Advanced... Check I1.0...' | German: 'S6 342 Row 35 Lost Advance Position... Check Ixxx.x German' | French: 'S6 342 Row 35 Lost Advance Position... Check Ixxx.x French'
  343 = 'Clamp Cylinder A1 Lost Returned... Check I1.1...' | German: 'S6 343 Row 35 Lost Return Position... Check Ixxx.x German' | French: 'S6 343 Row 35 Lost Return Position... Check Ixxx.x French'
  344 = 'Clamp Cylinder A1 Switch Fault... Check I1.0, I1.1...' | German: 'S6 344 Row 35 Switch Fault... Check Ixxx.x / Ixxx.x German' | French: 'S6 344 Row 35 Switch Fault... Check Ixxx.x / Ixxx.x French'
  345 = 'Spare' | German: 'S6 345 Row 35 Spare Message German' | French: 'S6 345 Row 35 Spare Message French'
  346 = 'Spare' | German: 'S6 346 Row 35 Spare Message German' | French: 'S6 346 Row 35 Spare Message French'
  347 = 'Spare' | German: 'S6 347 Row 35 Spare Message German' | French: 'S6 347 Row 35 Spare Message French'
  348 = 'Spare' | German: 'S6 348 Row 35 Spare Message German' | French: 'S6 348 Row 35 Spare Message French'
  349 = 'Spare' | German: 'S6 349 Row 35 Spare Message German' | French: 'S6 349 Row 35 Spare Message French'
  350 = 'Clamp Cylinder A1 Failed to Advance... Check Q1.0...' | German: 'S6 350 Row 36 Failed To Advance.. Check Qxxx.x German' | French: 'S6 350 Row 36 Failed To Advance.. Check Qxxx.x French'
  351 = 'Clamp Cylinder A1 Failed to Return... Check Q1.1...' | German: 'S6 351 Row 36 Failed To Return.. Check Qxxx.x German' | French: 'S6 351 Row 36 Failed To Return.. Check Qxxx.x French'
  352 = 'Clamp Cylinder A1 Lost Advanced... Check I1.0...' | German: 'S6 352 Row 36 Lost Advance Position... Check Ixxx.x German' | French: 'S6 352 Row 36 Lost Advance Position... Check Ixxx.x French'
  353 = 'Clamp Cylinder A1 Lost Returned... Check I1.1...' | German: 'S6 353 Row 36 Lost Return Position... Check Ixxx.x German' | French: 'S6 353 Row 36 Lost Return Position... Check Ixxx.x French'
  354 = 'Clamp Cylinder A1 Switch Fault... Check I1.0, I1.1...' | German: 'S6 354 Row 36 Switch Fault... Check Ixxx.x / Ixxx.x German' | French: 'S6 354 Row 36 Switch Fault... Check Ixxx.x / Ixxx.x French'
  355 = 'Spare' | German: 'S6 355 Row 36 Spare Message German' | French: 'S6 355 Row 36 Spare Message French'
  356 = 'Spare' | German: 'S6 356 Row 36 Spare Message German' | French: 'S6 356 Row 36 Spare Message French'
  357 = 'Spare' | German: 'S6 357 Row 36 Spare Message German' | French: 'S6 357 Row 36 Spare Message French'
  358 = 'Spare' | German: 'S6 358 Row 36 Spare Message German' | French: 'S6 358 Row 36 Spare Message French'
  359 = 'Spare' | German: 'S6 359 Row 36 Spare Message German' | French: 'S6 359 Row 36 Spare Message French'
  360 = 'Clamp Cylinder A1 Failed to Advance... Check Q1.0...' | German: 'S6 360 Row 37 Failed To Advance.. Check Qxxx.x German' | French: 'S6 360 Row 37 Failed To Advance.. Check Qxxx.x French'
  361 = 'Clamp Cylinder A1 Failed to Return... Check Q1.1...' | German: 'S6 361 Row 37 Failed To Return.. Check Qxxx.x German' | French: 'S6 361 Row 37 Failed To Return.. Check Qxxx.x French'
  362 = 'Clamp Cylinder A1 Lost Advanced... Check I1.0...' | German: 'S6 362 Row 37 Lost Advance Position... Check Ixxx.x German' | French: 'S6 362 Row 37 Lost Advance Position... Check Ixxx.x French'
  363 = 'Clamp Cylinder A1 Lost Returned... Check I1.1...' | German: 'S6 363 Row 37 Lost Return Position... Check Ixxx.x German' | French: 'S6 363 Row 37 Lost Return Position... Check Ixxx.x French'
  364 = 'Clamp Cylinder A1 Switch Fault... Check I1.0, I1.1...' | German: 'S6 364 Row 37 Switch Fault... Check Ixxx.x / Ixxx.x German' | French: 'S6 364 Row 37 Switch Fault... Check Ixxx.x / Ixxx.x French'
  365 = 'Spare' | German: 'S6 365 Row 37 Spare Message German' | French: 'S6 365 Row 37 Spare Message French'
  366 = 'Spare' | German: 'S6 366 Row 37 Spare Message German' | French: 'S6 366 Row 37 Spare Message French'
  367 = 'Spare' | German: 'S6 367 Row 37 Spare Message German' | French: 'S6 367 Row 37 Spare Message French'
  368 = 'Spare' | German: 'S6 368 Row 37 Spare Message German' | French: 'S6 368 Row 37 Spare Message French'
  369 = 'Spare' | German: 'S6 369 Row 37 Spare Message German' | French: 'S6 369 Row 37 Spare Message French'
  370 = 'Clamp Cylinder A1 Failed to Advance... Check Q1.0...' | German: 'S6 370 Row 38 Failed To Advance.. Check Qxxx.x German' | French: 'S6 370 Row 38 Failed To Advance.. Check Qxxx.x French'
  371 = 'Clamp Cylinder A1 Failed to Return... Check Q1.1...' | German: 'S6 371 Row 38 Failed To Return.. Check Qxxx.x German' | French: 'S6 371 Row 38 Failed To Return.. Check Qxxx.x French'
  372 = 'Clamp Cylinder A1 Lost Advanced... Check I1.0...' | German: 'S6 372 Row 38 Lost Advance Position... Check Ixxx.x German' | French: 'S6 372 Row 38 Lost Advance Position... Check Ixxx.x French'
  373 = 'Clamp Cylinder A1 Lost Returned... Check I1.1...' | German: 'S6 373 Row 38 Lost Return Position... Check Ixxx.x German' | French: 'S6 373 Row 38 Lost Return Position... Check Ixxx.x French'
  374 = 'Clamp Cylinder A1 Switch Fault... Check I1.0, I1.1...' | German: 'S6 374 Row 38 Switch Fault... Check Ixxx.x / Ixxx.x German' | French: 'S6 374 Row 38 Switch Fault... Check Ixxx.x / Ixxx.x French'
  375 = 'Spare' | German: 'S6 375 Row 38 Spare Message German' | French: 'S6 375 Row 38 Spare Message French'
  376 = 'Spare' | German: 'S6 376 Row 38 Spare Message German' | French: 'S6 376 Row 38 Spare Message French'
  377 = 'Spare' | German: 'S6 377 Row 38 Spare Message German' | French: 'S6 377 Row 38 Spare Message French'
  378 = 'Spare' | German: 'S6 378 Row 38 Spare Message German' | French: 'S6 378 Row 38 Spare Message French'
  379 = 'Spare' | German: 'S6 379 Row 38 Spare Message German' | French: 'S6 379 Row 38 Spare Message French'
  380 = 'Clamp Cylinder A1 Failed to Advance... Check Q1.0...' | German: 'S6 380 Row 39 Failed To Advance.. Check Qxxx.x German' | French: 'S6 380 Row 39 Failed To Advance.. Check Qxxx.x French'
  381 = 'Clamp Cylinder A1 Failed to Return... Check Q1.1...' | German: 'S6 381 Row 39 Failed To Return.. Check Qxxx.x German' | French: 'S6 381 Row 39 Failed To Return.. Check Qxxx.x French'
  382 = 'Clamp Cylinder A1 Lost Advanced... Check I1.0...' | German: 'S6 382 Row 39 Lost Advance Position... Check Ixxx.x German' | French: 'S6 382 Row 39 Lost Advance Position... Check Ixxx.x French'
  383 = 'Clamp Cylinder A1 Lost Returned... Check I1.1...' | German: 'S6 383 Row 39 Lost Return Position... Check Ixxx.x German' | French: 'S6 383 Row 39 Lost Return Position... Check Ixxx.x French'
  384 = 'Clamp Cylinder A1 Switch Fault... Check I1.0, I1.1...' | German: 'S6 384 Row 39 Switch Fault... Check Ixxx.x / Ixxx.x German' | French: 'S6 384 Row 39 Switch Fault... Check Ixxx.x / Ixxx.x French'
  385 = 'Spare' | German: 'S6 385 Row 39 Spare Message German' | French: 'S6 385 Row 39 Spare Message French'
  386 = 'Spare' | German: 'S6 386 Row 39 Spare Message German' | French: 'S6 386 Row 39 Spare Message French'
  387 = 'Spare' | German: 'S6 387 Row 39 Spare Message German' | French: 'S6 387 Row 39 Spare Message French'
  388 = 'Spare' | German: 'S6 388 Row 39 Spare Message German' | French: 'S6 388 Row 39 Spare Message French'
  389 = 'Spare' | German: 'S6 389 Row 39 Spare Message German' | French: 'S6 389 Row 39 Spare Message French'
  390 = 'Clamp Cylinder A1 Failed to Advance... Check Q1.0...' | German: 'S6 390 Row 40 Failed To Advance.. Check Qxxx.x German' | French: 'S6 390 Row 40 Failed To Advance.. Check Qxxx.x French'
  391 = 'Clamp Cylinder A1 Failed to Return... Check Q1.1...' | German: 'S6 391 Row 40 Failed To Return.. Check Qxxx.x German' | French: 'S6 391 Row 40 Failed To Return.. Check Qxxx.x French'
  392 = 'Clamp Cylinder A1 Lost Advanced... Check I1.0...' | German: 'S6 392 Row 40 Lost Advance Position... Check Ixxx.x German' | French: 'S6 392 Row 40 Lost Advance Position... Check Ixxx.x French'
  393 = 'Clamp Cylinder A1 Lost Returned... Check I1.1...' | German: 'S6 393 Row 40 Lost Return Position... Check Ixxx.x German' | French: 'S6 393 Row 40 Lost Return Position... Check Ixxx.x French'
  394 = 'Clamp Cylinder A1 Switch Fault... Check I1.0, I1.1...' | German: 'S6 394 Row 40 Switch Fault... Check Ixxx.x / Ixxx.x German' | French: 'S6 394 Row 40 Switch Fault... Check Ixxx.x / Ixxx.x French'
  395 = 'Spare' | German: 'S6 395 Row 40 Spare Message German' | French: 'S6 395 Row 40 Spare Message French'
  396 = 'Spare' | German: 'S6 396 Row 40 Spare Message German' | French: 'S6 396 Row 40 Spare Message French'
  397 = 'Spare' | German: 'S6 397 Row 40 Spare Message German' | French: 'S6 397 Row 40 Spare Message French'
  398 = 'Spare' | German: 'S6 398 Row 40 Spare Message German' | French: 'S6 398 Row 40 Spare Message French'
  399 = 'Spare' | German: 'S6 399 Row 40 Spare Message German' | French: 'S6 399 Row 40 Spare Message French'
  400 = 'Clamp Cylinder A1 Failed to Advance... Check Q1.0...' | German: 'S6 400 Row 41 Failed To Advance.. Check Qxxx.x German' | French: 'S6 400 Row 41 Failed To Advance.. Check Qxxx.x French'
  401 = 'Clamp Cylinder A1 Failed to Return... Check Q1.1...' | German: 'S6 401 Row 41 Failed To Return.. Check Qxxx.x German' | French: 'S6 401 Row 41 Failed To Return.. Check Qxxx.x French'
  402 = 'Clamp Cylinder A1 Lost Advanced... Check I1.0...' | German: 'S6 402 Row 41 Lost Advance Position... Check Ixxx.x German' | French: 'S6 402 Row 41 Lost Advance Position... Check Ixxx.x French'
  403 = 'Clamp Cylinder A1 Lost Returned... Check I1.1...' | German: 'S6 403 Row 41 Lost Return Position... Check Ixxx.x German' | French: 'S6 403 Row 41 Lost Return Position... Check Ixxx.x French'
  404 = 'Clamp Cylinder A1 Switch Fault... Check I1.0, I1.1...' | German: 'S6 404 Row 41 Switch Fault... Check Ixxx.x / Ixxx.x German' | French: 'S6 404 Row 41 Switch Fault... Check Ixxx.x / Ixxx.x French'
  405 = 'Spare' | German: 'S6 405 Row 41 Spare Message German' | French: 'S6 405 Row 41 Spare Message French'
  406 = 'Spare' | German: 'S6 406 Row 41 Spare Message German' | French: 'S6 406 Row 41 Spare Message French'
  407 = 'Spare' | German: 'S6 407 Row 41 Spare Message German' | French: 'S6 407 Row 41 Spare Message French'
  408 = 'Spare' | German: 'S6 408 Row 41 Spare Message German' | French: 'S6 408 Row 41 Spare Message French'
  409 = 'Spare' | German: 'S6 409 Row 41 Spare Message German' | French: 'S6 409 Row 41 Spare Message French'
  410 = 'Clamp Cylinder A1 Failed to Advance... Check Q1.0...' | German: 'S6 410 Row 42 Failed To Advance.. Check Qxxx.x German' | French: 'S6 410 Row 42 Failed To Advance.. Check Qxxx.x French'
  411 = 'Clamp Cylinder A1 Failed to Return... Check Q1.1...' | German: 'S6 411 Row 42 Failed To Return.. Check Qxxx.x German' | French: 'S6 411 Row 42 Failed To Return.. Check Qxxx.x French'
  412 = 'Clamp Cylinder A1 Lost Advanced... Check I1.0...' | German: 'S6 412 Row 42 Lost Advance Position... Check Ixxx.x German' | French: 'S6 412 Row 42 Lost Advance Position... Check Ixxx.x French'
  413 = 'Clamp Cylinder A1 Lost Returned... Check I1.1...' | German: 'S6 413 Row 42 Lost Return Position... Check Ixxx.x German' | French: 'S6 413 Row 42 Lost Return Position... Check Ixxx.x French'
  414 = 'Clamp Cylinder A1 Switch Fault... Check I1.0, I1.1...' | German: 'S6 414 Row 42 Switch Fault... Check Ixxx.x / Ixxx.x German' | French: 'S6 414 Row 42 Switch Fault... Check Ixxx.x / Ixxx.x French'
  415 = 'Spare' | German: 'S6 415 Row 42 Spare Message German' | French: 'S6 415 Row 42 Spare Message French'
  416 = 'Spare' | German: 'S6 416 Row 42 Spare Message German' | French: 'S6 416 Row 42 Spare Message French'
  417 = 'Spare' | German: 'S6 417 Row 42 Spare Message German' | French: 'S6 417 Row 42 Spare Message French'
  418 = 'Spare' | German: 'S6 418 Row 42 Spare Message German' | French: 'S6 418 Row 42 Spare Message French'
  419 = 'Spare' | German: 'S6 419 Row 42 Spare Message German' | French: 'S6 419 Row 42 Spare Message French'
  420 = 'Clamp Cylinder A1 Failed to Advance... Check Q1.0...' | German: 'S6 420 Row 43 Failed To Advance.. Check Qxxx.x German' | French: 'S6 420 Row 43 Failed To Advance.. Check Qxxx.x French'
  421 = 'Clamp Cylinder A1 Failed to Return... Check Q1.1...' | German: 'S6 421 Row 43 Failed To Return.. Check Qxxx.x German' | French: 'S6 421 Row 43 Failed To Return.. Check Qxxx.x French'
  422 = 'Clamp Cylinder A1 Lost Advanced... Check I1.0...' | German: 'S6 422 Row 43 Lost Advance Position... Check Ixxx.x German' | French: 'S6 422 Row 43 Lost Advance Position... Check Ixxx.x French'
  423 = 'Clamp Cylinder A1 Lost Returned... Check I1.1...' | German: 'S6 423 Row 43 Lost Return Position... Check Ixxx.x German' | French: 'S6 423 Row 43 Lost Return Position... Check Ixxx.x French'
  424 = 'Clamp Cylinder A1 Switch Fault... Check I1.0, I1.1...' | German: 'S6 424 Row 43 Switch Fault... Check Ixxx.x / Ixxx.x German' | French: 'S6 424 Row 43 Switch Fault... Check Ixxx.x / Ixxx.x French'
  425 = 'Spare' | German: 'S6 425 Row 43 Spare Message German' | French: 'S6 425 Row 43 Spare Message French'
  426 = 'Spare' | German: 'S6 426 Row 43 Spare Message German' | French: 'S6 426 Row 43 Spare Message French'
  427 = 'Spare' | German: 'S6 427 Row 43 Spare Message German' | French: 'S6 427 Row 43 Spare Message French'
  428 = 'Spare' | German: 'S6 428 Row 43 Spare Message German' | French: 'S6 428 Row 43 Spare Message French'
  429 = 'Spare' | German: 'S6 429 Row 43 Spare Message German' | French: 'S6 429 Row 43 Spare Message French'
  430 = 'Clamp Cylinder A1 Failed to Advance... Check Q1.0...' | German: 'S6 430 Row 44 Failed To Advance.. Check Qxxx.x German' | French: 'S6 430 Row 44 Failed To Advance.. Check Qxxx.x French'
  431 = 'Clamp Cylinder A1 Failed to Return... Check Q1.1...' | German: 'S6 431 Row 44 Failed To Return.. Check Qxxx.x German' | French: 'S6 431 Row 44 Failed To Return.. Check Qxxx.x French'
  432 = 'Clamp Cylinder A1 Lost Advanced... Check I1.0...' | German: 'S6 432 Row 44 Lost Advance Position... Check Ixxx.x German' | French: 'S6 432 Row 44 Lost Advance Position... Check Ixxx.x French'
  433 = 'Clamp Cylinder A1 Lost Returned... Check I1.1...' | German: 'S6 433 Row 44 Lost Return Position... Check Ixxx.x German' | French: 'S6 433 Row 44 Lost Return Position... Check Ixxx.x French'
  434 = 'Clamp Cylinder A1 Switch Fault... Check I1.0, I1.1...' | German: 'S6 434 Row 44 Switch Fault... Check Ixxx.x / Ixxx.x German' | French: 'S6 434 Row 44 Switch Fault... Check Ixxx.x / Ixxx.x French'
  435 = 'Spare' | German: 'S6 435 Row 44 Spare Message German' | French: 'S6 435 Row 44 Spare Message French'
  436 = 'Spare' | German: 'S6 436 Row 44 Spare Message German' | French: 'S6 436 Row 44 Spare Message French'
  437 = 'Spare' | German: 'S6 437 Row 44 Spare Message German' | French: 'S6 437 Row 44 Spare Message French'
  438 = 'Spare' | German: 'S6 438 Row 44 Spare Message German' | French: 'S6 438 Row 44 Spare Message French'
  439 = 'Spare' | German: 'S6 439 Row 44 Spare Message German' | French: 'S6 439 Row 44 Spare Message French'
  440 = 'Clamp Cylinder A1 Failed to Advance... Check Q1.0...' | German: 'S6 440 Row 45 Failed To Advance.. Check Qxxx.x German' | French: 'S6 440 Row 45 Failed To Advance.. Check Qxxx.x French'
  441 = 'Clamp Cylinder A1 Failed to Return... Check Q1.1...' | German: 'S6 441 Row 45 Failed To Return.. Check Qxxx.x German' | French: 'S6 441 Row 45 Failed To Return.. Check Qxxx.x French'
  442 = 'Clamp Cylinder A1 Lost Advanced... Check I1.0...' | German: 'S6 442 Row 45 Lost Advance Position... Check Ixxx.x German' | French: 'S6 442 Row 45 Lost Advance Position... Check Ixxx.x French'
  443 = 'Clamp Cylinder A1 Lost Returned... Check I1.1...' | German: 'S6 443 Row 45 Lost Return Position... Check Ixxx.x German' | French: 'S6 443 Row 45 Lost Return Position... Check Ixxx.x French'
  444 = 'Clamp Cylinder A1 Switch Fault... Check I1.0, I1.1...' | German: 'S6 444 Row 45 Switch Fault... Check Ixxx.x / Ixxx.x German' | French: 'S6 444 Row 45 Switch Fault... Check Ixxx.x / Ixxx.x French'
  445 = 'Spare' | German: 'S6 445 Row 45 Spare Message German' | French: 'S6 445 Row 45 Spare Message French'
  446 = 'Spare' | German: 'S6 446 Row 45 Spare Message German' | French: 'S6 446 Row 45 Spare Message French'
  447 = 'Spare' | German: 'S6 447 Row 45 Spare Message German' | French: 'S6 447 Row 45 Spare Message French'
  448 = 'Spare' | German: 'S6 448 Row 45 Spare Message German' | French: 'S6 448 Row 45 Spare Message French'
  449 = 'Spare' | German: 'S6 449 Row 45 Spare Message German' | French: 'S6 449 Row 45 Spare Message French'
  450 = 'Clamp Cylinder A1 Failed to Advance... Check Q1.0...' | German: 'S6 450 Row 46 Failed To Advance.. Check Qxxx.x German' | French: 'S6 450 Row 46 Failed To Advance.. Check Qxxx.x French'
  451 = 'Clamp Cylinder A1 Failed to Return... Check Q1.1...' | German: 'S6 451 Row 46 Failed To Return.. Check Qxxx.x German' | French: 'S6 451 Row 46 Failed To Return.. Check Qxxx.x French'
  452 = 'Clamp Cylinder A1 Lost Advanced... Check I1.0...' | German: 'S6 452 Row 46 Lost Advance Position... Check Ixxx.x German' | French: 'S6 452 Row 46 Lost Advance Position... Check Ixxx.x French'
  453 = 'Clamp Cylinder A1 Lost Returned... Check I1.1...' | German: 'S6 453 Row 46 Lost Return Position... Check Ixxx.x German' | French: 'S6 453 Row 46 Lost Return Position... Check Ixxx.x French'
  454 = 'Clamp Cylinder A1 Switch Fault... Check I1.0, I1.1...' | German: 'S6 454 Row 46 Switch Fault... Check Ixxx.x / Ixxx.x German' | French: 'S6 454 Row 46 Switch Fault... Check Ixxx.x / Ixxx.x French'
  455 = 'Spare' | German: 'S6 455 Row 46 Spare Message German' | French: 'S6 455 Row 46 Spare Message French'
  456 = 'Spare' | German: 'S6 456 Row 46 Spare Message German' | French: 'S6 456 Row 46 Spare Message French'
  457 = 'Spare' | German: 'S6 457 Row 46 Spare Message German' | French: 'S6 457 Row 46 Spare Message French'
  458 = 'Spare' | German: 'S6 458 Row 46 Spare Message German' | French: 'S6 458 Row 46 Spare Message French'
  459 = 'Spare' | German: 'S6 459 Row 46 Spare Message German' | French: 'S6 459 Row 46 Spare Message French'
  460 = 'Clamp Cylinder A1 Failed to Advance... Check Q1.0...' | German: 'S6 460 Row 47 Failed To Advance.. Check Qxxx.x German' | French: 'S6 460 Row 47 Failed To Advance.. Check Qxxx.x French'
  461 = 'Clamp Cylinder A1 Failed to Return... Check Q1.1...' | German: 'S6 461 Row 47 Failed To Return.. Check Qxxx.x German' | French: 'S6 461 Row 47 Failed To Return.. Check Qxxx.x French'
  462 = 'Clamp Cylinder A1 Lost Advanced... Check I1.0...' | German: 'S6 462 Row 47 Lost Advance Position... Check Ixxx.x German' | French: 'S6 462 Row 47 Lost Advance Position... Check Ixxx.x French'
  463 = 'Clamp Cylinder A1 Lost Returned... Check I1.1...' | German: 'S6 463 Row 47 Lost Return Position... Check Ixxx.x German' | French: 'S6 463 Row 47 Lost Return Position... Check Ixxx.x French'
  464 = 'Clamp Cylinder A1 Switch Fault... Check I1.0, I1.1...' | German: 'S6 464 Row 47 Switch Fault... Check Ixxx.x / Ixxx.x German' | French: 'S6 464 Row 47 Switch Fault... Check Ixxx.x / Ixxx.x French'
  465 = 'Spare' | German: 'S6 465 Row 47 Spare Message German' | French: 'S6 465 Row 47 Spare Message French'
  466 = 'Spare' | German: 'S6 466 Row 47 Spare Message German' | French: 'S6 466 Row 47 Spare Message French'
  467 = 'Spare' | German: 'S6 467 Row 47 Spare Message German' | French: 'S6 467 Row 47 Spare Message French'
  468 = 'Spare' | German: 'S6 468 Row 47 Spare Message German' | French: 'S6 468 Row 47 Spare Message French'
  469 = 'Spare' | German: 'S6 469 Row 47 Spare Message German' | French: 'S6 469 Row 47 Spare Message French'
  470 = 'Clamp Cylinder A1 Failed to Advance... Check Q1.0...' | German: 'S6 470 Row 48 Failed To Advance.. Check Qxxx.x German' | French: 'S6 470 Row 48 Failed To Advance.. Check Qxxx.x French'
  471 = 'Clamp Cylinder A1 Failed to Return... Check Q1.1...' | German: 'S6 471 Row 48 Failed To Return.. Check Qxxx.x German' | French: 'S6 471 Row 48 Failed To Return.. Check Qxxx.x French'
  472 = 'Clamp Cylinder A1 Lost Advanced... Check I1.0...' | German: 'S6 472 Row 48 Lost Advance Position... Check Ixxx.x German' | French: 'S6 472 Row 48 Lost Advance Position... Check Ixxx.x French'
  473 = 'Clamp Cylinder A1 Lost Returned... Check I1.1...' | German: 'S6 473 Row 48 Lost Return Position... Check Ixxx.x German' | French: 'S6 473 Row 48 Lost Return Position... Check Ixxx.x French'
  474 = 'Clamp Cylinder A1 Switch Fault... Check I1.0, I1.1...' | German: 'S6 474 Row 48 Switch Fault... Check Ixxx.x / Ixxx.x German' | French: 'S6 474 Row 48 Switch Fault... Check Ixxx.x / Ixxx.x French'
  475 = 'Spare' | German: 'S6 475 Row 48 Spare Message German' | French: 'S6 475 Row 48 Spare Message French'
  476 = 'Spare' | German: 'S6 476 Row 48 Spare Message German' | French: 'S6 476 Row 48 Spare Message French'
  477 = 'Spare' | German: 'S6 477 Row 48 Spare Message German' | French: 'S6 477 Row 48 Spare Message French'
  478 = 'Spare' | German: 'S6 478 Row 48 Spare Message German' | French: 'S6 478 Row 48 Spare Message French'
  479 = 'Spare' | German: 'S6 479 Row 48 Spare Message German' | French: 'S6 479 Row 48 Spare Message French'
  480 = 'Clamp Cylinder A1 Failed to Advance... Check Q1.0...' | German: 'S6 480 Row 49 Failed To Advance.. Check Qxxx.x German' | French: 'S6 480 Row 49 Failed To Advance.. Check Qxxx.x French'
  481 = 'Clamp Cylinder A1 Failed to Return... Check Q1.1...' | German: 'S6 481 Row 49 Failed To Return.. Check Qxxx.x German' | French: 'S6 481 Row 49 Failed To Return.. Check Qxxx.x French'
  482 = 'Clamp Cylinder A1 Lost Advanced... Check I1.0...' | German: 'S6 482 Row 49 Lost Advance Position... Check Ixxx.x German' | French: 'S6 482 Row 49 Lost Advance Position... Check Ixxx.x French'
  483 = 'Clamp Cylinder A1 Lost Returned... Check I1.1...' | German: 'S6 483 Row 49 Lost Return Position... Check Ixxx.x German' | French: 'S6 483 Row 49 Lost Return Position... Check Ixxx.x French'
  484 = 'Clamp Cylinder A1 Switch Fault... Check I1.0, I1.1...' | German: 'S6 484 Row 49 Switch Fault... Check Ixxx.x / Ixxx.x German' | French: 'S6 484 Row 49 Switch Fault... Check Ixxx.x / Ixxx.x French'
  485 = 'Spare' | German: 'S6 485 Row 49 Spare Message German' | French: 'S6 485 Row 49 Spare Message French'
  486 = 'Spare' | German: 'S6 486 Row 49 Spare Message German' | French: 'S6 486 Row 49 Spare Message French'
  487 = 'Spare' | German: 'S6 487 Row 49 Spare Message German' | French: 'S6 487 Row 49 Spare Message French'
  488 = 'Spare' | German: 'S6 488 Row 49 Spare Message German' | French: 'S6 488 Row 49 Spare Message French'
  489 = 'Spare' | German: 'S6 489 Row 49 Spare Message German' | French: 'S6 489 Row 49 Spare Message French'
  490 = 'Clamp Cylinder A1 Failed to Advance... Check Q1.0...' | German: 'S6 490 Row 50 Failed To Advance.. Check Qxxx.x German' | French: 'S6 490 Row 50 Failed To Advance.. Check Qxxx.x French'
  491 = 'Clamp Cylinder A1 Failed to Return... Check Q1.1...' | German: 'S6 491 Row 50 Failed To Return.. Check Qxxx.x German' | French: 'S6 491 Row 50 Failed To Return.. Check Qxxx.x French'
  492 = 'Clamp Cylinder A1 Lost Advanced... Check I1.0...' | German: 'S6 492 Row 50 Lost Advance Position... Check Ixxx.x German' | French: 'S6 492 Row 50 Lost Advance Position... Check Ixxx.x French'
  493 = 'Clamp Cylinder A1 Lost Returned... Check I1.1...' | German: 'S6 493 Row 50 Lost Return Position... Check Ixxx.x German' | French: 'S6 493 Row 50 Lost Return Position... Check Ixxx.x French'
  494 = 'Clamp Cylinder A1 Switch Fault... Check I1.0, I1.1...' | German: 'S6 494 Row 50 Switch Fault... Check Ixxx.x / Ixxx.x German' | French: 'S6 494 Row 50 Switch Fault... Check Ixxx.x / Ixxx.x French'
  495 = 'Spare' | German: 'S6 495 Row 50 Spare Message German' | French: 'S6 495 Row 50 Spare Message French'
  496 = 'Spare' | German: 'S6 496 Row 50 Spare Message German' | French: 'S6 496 Row 50 Spare Message French'
  497 = 'Spare' | German: 'S6 497 Row 50 Spare Message German' | French: 'S6 497 Row 50 Spare Message French'
  498 = 'Spare' | German: 'S6 498 Row 50 Spare Message German' | French: 'S6 498 Row 50 Spare Message French'
  499 = 'Spare' | German: 'S6 499 Row 50 Spare Message German' | French: 'S6 499 Row 50 Spare Message French'
  500 = 'Clamp Cylinder A1 Failed to Advance... Check Q1.0...' | German: 'S6 500 Row 51 Failed To Advance.. Check Qxxx.x German' | French: 'S6 500 Row 51 Failed To Advance.. Check Qxxx.x French'
  501 = 'Clamp Cylinder A1 Failed to Return... Check Q1.1...' | German: 'S6 501 Row 51 Failed To Return.. Check Qxxx.x German' | French: 'S6 501 Row 51 Failed To Return.. Check Qxxx.x French'
  502 = 'Clamp Cylinder A1 Lost Advanced... Check I1.0...' | German: 'S6 502 Row 51 Lost Advance Position... Check Ixxx.x German' | French: 'S6 502 Row 51 Lost Advance Position... Check Ixxx.x French'
  503 = 'Clamp Cylinder A1 Lost Returned... Check I1.1...' | German: 'S6 503 Row 51 Lost Return Position... Check Ixxx.x German' | French: 'S6 503 Row 51 Lost Return Position... Check Ixxx.x French'
  504 = 'Clamp Cylinder A1 Switch Fault... Check I1.0, I1.1...' | German: 'S6 504 Row 51 Switch Fault... Check Ixxx.x / Ixxx.x German' | French: 'S6 504 Row 51 Switch Fault... Check Ixxx.x / Ixxx.x French'
  505 = 'Spare' | German: 'S6 505 Row 51 Spare Message German' | French: 'S6 505 Row 51 Spare Message French'
  506 = 'Spare' | German: 'S6 506 Row 51 Spare Message German' | French: 'S6 506 Row 51 Spare Message French'
  507 = 'Spare' | German: 'S6 507 Row 51 Spare Message German' | French: 'S6 507 Row 51 Spare Message French'
  508 = 'Spare' | German: 'S6 508 Row 51 Spare Message German' | French: 'S6 508 Row 51 Spare Message French'
  509 = 'Spare' | German: 'S6 509 Row 51 Spare Message German' | French: 'S6 509 Row 51 Spare Message French'
  510 = 'Clamp Cylinder A1 Failed to Advance... Check Q1.0...' | German: 'S6 510 Row 52 Failed To Advance.. Check Qxxx.x German' | French: 'S6 510 Row 52 Failed To Advance.. Check Qxxx.x French'
  511 = 'Clamp Cylinder A1 Failed to Return... Check Q1.1...' | German: 'S6 511 Row 52 Failed To Return.. Check Qxxx.x German' | French: 'S6 511 Row 52 Failed To Return.. Check Qxxx.x French'
  512 = 'Clamp Cylinder A1 Lost Advanced... Check I1.0...' | German: 'S6 512 Row 52 Lost Advance Position... Check Ixxx.x German' | French: 'S6 512 Row 52 Lost Advance Position... Check Ixxx.x French'
  513 = 'Clamp Cylinder A1 Lost Returned... Check I1.1...' | German: 'S6 513 Row 52 Lost Return Position... Check Ixxx.x German' | French: 'S6 513 Row 52 Lost Return Position... Check Ixxx.x French'
  514 = 'Clamp Cylinder A1 Switch Fault... Check I1.0, I1.1...' | German: 'S6 514 Row 52 Switch Fault... Check Ixxx.x / Ixxx.x German' | French: 'S6 514 Row 52 Switch Fault... Check Ixxx.x / Ixxx.x French'
  515 = 'Spare' | German: 'S6 515 Row 52 Spare Message German' | French: 'S6 515 Row 52 Spare Message French'
  516 = 'Spare' | German: 'S6 516 Row 52 Spare Message German' | French: 'S6 516 Row 52 Spare Message French'
  517 = 'Spare' | German: 'S6 517 Row 52 Spare Message German' | French: 'S6 517 Row 52 Spare Message French'
  518 = 'Spare' | German: 'S6 518 Row 52 Spare Message German' | French: 'S6 518 Row 52 Spare Message French'
  519 = 'Spare' | German: 'S6 519 Row 52 Spare Message German' | French: 'S6 519 Row 52 Spare Message French'
  520 = 'Clamp Cylinder A1 Failed to Advance... Check Q1.0...' | German: 'S6 520 Row 53 Failed To Advance.. Check Qxxx.x German' | French: 'S6 520 Row 53 Failed To Advance.. Check Qxxx.x French'
  521 = 'Clamp Cylinder A1 Failed to Return... Check Q1.1...' | German: 'S6 521 Row 53 Failed To Return.. Check Qxxx.x German' | French: 'S6 521 Row 53 Failed To Return.. Check Qxxx.x French'
  522 = 'Clamp Cylinder A1 Lost Advanced... Check I1.0...' | German: 'S6 522 Row 53 Lost Advance Position... Check Ixxx.x German' | French: 'S6 522 Row 53 Lost Advance Position... Check Ixxx.x French'
  523 = 'Clamp Cylinder A1 Lost Returned... Check I1.1...' | German: 'S6 523 Row 53 Lost Return Position... Check Ixxx.x German' | French: 'S6 523 Row 53 Lost Return Position... Check Ixxx.x French'
  524 = 'Clamp Cylinder A1 Switch Fault... Check I1.0, I1.1...' | German: 'S6 524 Row 53 Switch Fault... Check Ixxx.x / Ixxx.x German' | French: 'S6 524 Row 53 Switch Fault... Check Ixxx.x / Ixxx.x French'
  525 = 'Spare' | German: 'S6 525 Row 53 Spare Message German' | French: 'S6 525 Row 53 Spare Message French'
  526 = 'Spare' | German: 'S6 526 Row 53 Spare Message German' | French: 'S6 526 Row 53 Spare Message French'
  527 = 'Spare' | German: 'S6 527 Row 53 Spare Message German' | French: 'S6 527 Row 53 Spare Message French'
  528 = 'Spare' | German: 'S6 528 Row 53 Spare Message German' | French: 'S6 528 Row 53 Spare Message French'
  529 = 'Spare' | German: 'S6 529 Row 53 Spare Message German' | French: 'S6 529 Row 53 Spare Message French'
  530 = 'Clamp Cylinder A1 Failed to Advance... Check Q1.0...' | German: 'S6 530 Row 54 Failed To Advance.. Check Qxxx.x German' | French: 'S6 530 Row 54 Failed To Advance.. Check Qxxx.x French'
  531 = 'Clamp Cylinder A1 Failed to Return... Check Q1.1...' | German: 'S6 531 Row 54 Failed To Return.. Check Qxxx.x German' | French: 'S6 531 Row 54 Failed To Return.. Check Qxxx.x French'
  532 = 'Clamp Cylinder A1 Lost Advanced... Check I1.0...' | German: 'S6 532 Row 54 Lost Advance Position... Check Ixxx.x German' | French: 'S6 532 Row 54 Lost Advance Position... Check Ixxx.x French'
  533 = 'Clamp Cylinder A1 Lost Returned... Check I1.1...' | German: 'S6 533 Row 54 Lost Return Position... Check Ixxx.x German' | French: 'S6 533 Row 54 Lost Return Position... Check Ixxx.x French'
  534 = 'Clamp Cylinder A1 Switch Fault... Check I1.0, I1.1...' | German: 'S6 534 Row 54 Switch Fault... Check Ixxx.x / Ixxx.x German' | French: 'S6 534 Row 54 Switch Fault... Check Ixxx.x / Ixxx.x French'
  535 = 'Spare' | German: 'S6 535 Row 54 Spare Message German' | French: 'S6 535 Row 54 Spare Message French'
  536 = 'Spare' | German: 'S6 536 Row 54 Spare Message German' | French: 'S6 536 Row 54 Spare Message French'
  537 = 'Spare' | German: 'S6 537 Row 54 Spare Message German' | French: 'S6 537 Row 54 Spare Message French'
  538 = 'Spare' | German: 'S6 538 Row 54 Spare Message German' | French: 'S6 538 Row 54 Spare Message French'
  539 = 'Spare' | German: 'S6 539 Row 54 Spare Message German' | French: 'S6 539 Row 54 Spare Message French'
  540 = 'Clamp Cylinder A1 Failed to Advance... Check Q1.0...' | German: 'S6 540 Row 55 Failed To Advance.. Check Qxxx.x German' | French: 'S6 540 Row 55 Failed To Advance.. Check Qxxx.x French'
  541 = 'Clamp Cylinder A1 Failed to Return... Check Q1.1...' | German: 'S6 541 Row 55 Failed To Return.. Check Qxxx.x German' | French: 'S6 541 Row 55 Failed To Return.. Check Qxxx.x French'
  542 = 'Clamp Cylinder A1 Lost Advanced... Check I1.0...' | German: 'S6 542 Row 55 Lost Advance Position... Check Ixxx.x German' | French: 'S6 542 Row 55 Lost Advance Position... Check Ixxx.x French'
  543 = 'Clamp Cylinder A1 Lost Returned... Check I1.1...' | German: 'S6 543 Row 55 Lost Return Position... Check Ixxx.x German' | French: 'S6 543 Row 55 Lost Return Position... Check Ixxx.x French'
  544 = 'Clamp Cylinder A1 Switch Fault... Check I1.0, I1.1...' | German: 'S6 544 Row 55 Switch Fault... Check Ixxx.x / Ixxx.x German' | French: 'S6 544 Row 55 Switch Fault... Check Ixxx.x / Ixxx.x French'
  545 = 'Spare' | German: 'S6 545 Row 55 Spare Message German' | French: 'S6 545 Row 55 Spare Message French'
  546 = 'Spare' | German: 'S6 546 Row 55 Spare Message German' | French: 'S6 546 Row 55 Spare Message French'
  547 = 'Spare' | German: 'S6 547 Row 55 Spare Message German' | French: 'S6 547 Row 55 Spare Message French'
  548 = 'Spare' | German: 'S6 548 Row 55 Spare Message German' | French: 'S6 548 Row 55 Spare Message French'
  549 = 'Spare' | German: 'S6 549 Row 55 Spare Message German' | French: 'S6 549 Row 55 Spare Message French'
  550 = 'Clamp Cylinder A1 Failed to Advance... Check Q1.0...' | German: 'S6 550 Row 56 Failed To Advance.. Check Qxxx.x German' | French: 'S6 550 Row 56 Failed To Advance.. Check Qxxx.x French'
  551 = 'Clamp Cylinder A1 Failed to Return... Check Q1.1...' | German: 'S6 551 Row 56 Failed To Return.. Check Qxxx.x German' | French: 'S6 551 Row 56 Failed To Return.. Check Qxxx.x French'
  552 = 'Clamp Cylinder A1 Lost Advanced... Check I1.0...' | German: 'S6 552 Row 56 Lost Advance Position... Check Ixxx.x German' | French: 'S6 552 Row 56 Lost Advance Position... Check Ixxx.x French'
  553 = 'Clamp Cylinder A1 Lost Returned... Check I1.1...' | German: 'S6 553 Row 56 Lost Return Position... Check Ixxx.x German' | French: 'S6 553 Row 56 Lost Return Position... Check Ixxx.x French'
  554 = 'Clamp Cylinder A1 Switch Fault... Check I1.0, I1.1...' | German: 'S6 554 Row 56 Switch Fault... Check Ixxx.x / Ixxx.x German' | French: 'S6 554 Row 56 Switch Fault... Check Ixxx.x / Ixxx.x French'
  555 = 'Spare' | German: 'S6 555 Row 56 Spare Message German' | French: 'S6 555 Row 56 Spare Message French'
  556 = 'Spare' | German: 'S6 556 Row 56 Spare Message German' | French: 'S6 556 Row 56 Spare Message French'
  557 = 'Spare' | German: 'S6 557 Row 56 Spare Message German' | French: 'S6 557 Row 56 Spare Message French'
  558 = 'Spare' | German: 'S6 558 Row 56 Spare Message German' | French: 'S6 558 Row 56 Spare Message French'
  559 = 'Spare' | German: 'S6 559 Row 56 Spare Message German' | French: 'S6 559 Row 56 Spare Message French'
  560 = 'Clamp Cylinder A1 Failed to Advance... Check Q1.0...' | German: 'S6 560 Row 57 Failed To Advance.. Check Qxxx.x German' | French: 'S6 560 Row 57 Failed To Advance.. Check Qxxx.x French'
  561 = 'Clamp Cylinder A1 Failed to Return... Check Q1.1...' | German: 'S6 561 Row 57 Failed To Return.. Check Qxxx.x German' | French: 'S6 561 Row 57 Failed To Return.. Check Qxxx.x French'
  562 = 'Clamp Cylinder A1 Lost Advanced... Check I1.0...' | German: 'S6 562 Row 57 Lost Advance Position... Check Ixxx.x German' | French: 'S6 562 Row 57 Lost Advance Position... Check Ixxx.x French'
  563 = 'Clamp Cylinder A1 Lost Returned... Check I1.1...' | German: 'S6 563 Row 57 Lost Return Position... Check Ixxx.x German' | French: 'S6 563 Row 57 Lost Return Position... Check Ixxx.x French'
  564 = 'Clamp Cylinder A1 Switch Fault... Check I1.0, I1.1...' | German: 'S6 564 Row 57 Switch Fault... Check Ixxx.x / Ixxx.x German' | French: 'S6 564 Row 57 Switch Fault... Check Ixxx.x / Ixxx.x French'
  565 = 'Spare' | German: 'S6 565 Row 57 Spare Message German' | French: 'S6 565 Row 57 Spare Message French'
  566 = 'Spare' | German: 'S6 566 Row 57 Spare Message German' | French: 'S6 566 Row 57 Spare Message French'
  567 = 'Spare' | German: 'S6 567 Row 57 Spare Message German' | French: 'S6 567 Row 57 Spare Message French'
  568 = 'Spare' | German: 'S6 568 Row 57 Spare Message German' | French: 'S6 568 Row 57 Spare Message French'
  569 = 'Spare' | German: 'S6 569 Row 57 Spare Message German' | French: 'S6 569 Row 57 Spare Message French'
  570 = 'Clamp Cylinder A1 Failed to Advance... Check Q1.0...' | German: 'S6 570 Row 58 Failed To Advance.. Check Qxxx.x German' | French: 'S6 570 Row 58 Failed To Advance.. Check Qxxx.x French'
  571 = 'Clamp Cylinder A1 Failed to Return... Check Q1.1...' | German: 'S6 571 Row 58 Failed To Return.. Check Qxxx.x German' | French: 'S6 571 Row 58 Failed To Return.. Check Qxxx.x French'
  572 = 'Clamp Cylinder A1 Lost Advanced... Check I1.0...' | German: 'S6 572 Row 58 Lost Advance Position... Check Ixxx.x German' | French: 'S6 572 Row 58 Lost Advance Position... Check Ixxx.x French'
  573 = 'Clamp Cylinder A1 Lost Returned... Check I1.1...' | German: 'S6 573 Row 58 Lost Return Position... Check Ixxx.x German' | French: 'S6 573 Row 58 Lost Return Position... Check Ixxx.x French'
  574 = 'Clamp Cylinder A1 Switch Fault... Check I1.0, I1.1...' | German: 'S6 574 Row 58 Switch Fault... Check Ixxx.x / Ixxx.x German' | French: 'S6 574 Row 58 Switch Fault... Check Ixxx.x / Ixxx.x French'
  575 = 'Spare' | German: 'S6 575 Row 58 Spare Message German' | French: 'S6 575 Row 58 Spare Message French'
  576 = 'Spare' | German: 'S6 576 Row 58 Spare Message German' | French: 'S6 576 Row 58 Spare Message French'
  577 = 'Spare' | German: 'S6 577 Row 58 Spare Message German' | French: 'S6 577 Row 58 Spare Message French'
  578 = 'Spare' | German: 'S6 578 Row 58 Spare Message German' | French: 'S6 578 Row 58 Spare Message French'
  579 = 'Spare' | German: 'S6 579 Row 58 Spare Message German' | French: 'S6 579 Row 58 Spare Message French'
  580 = 'Clamp Cylinder A1 Failed to Advance... Check Q1.0...' | German: 'S6 580 Row 59 Failed To Advance.. Check Qxxx.x German' | French: 'S6 580 Row 59 Failed To Advance.. Check Qxxx.x French'
  581 = 'Clamp Cylinder A1 Failed to Return... Check Q1.1...' | German: 'S6 581 Row 59 Failed To Return.. Check Qxxx.x German' | French: 'S6 581 Row 59 Failed To Return.. Check Qxxx.x French'
  582 = 'Clamp Cylinder A1 Lost Advanced... Check I1.0...' | German: 'S6 582 Row 59 Lost Advance Position... Check Ixxx.x German' | French: 'S6 582 Row 59 Lost Advance Position... Check Ixxx.x French'
  583 = 'Clamp Cylinder A1 Lost Returned... Check I1.1...' | German: 'S6 583 Row 59 Lost Return Position... Check Ixxx.x German' | French: 'S6 583 Row 59 Lost Return Position... Check Ixxx.x French'
  584 = 'Clamp Cylinder A1 Switch Fault... Check I1.0, I1.1...' | German: 'S6 584 Row 59 Switch Fault... Check Ixxx.x / Ixxx.x German' | French: 'S6 584 Row 59 Switch Fault... Check Ixxx.x / Ixxx.x French'
  585 = 'Spare' | German: 'S6 585 Row 59 Spare Message German' | French: 'S6 585 Row 59 Spare Message French'
  586 = 'Spare' | German: 'S6 586 Row 59 Spare Message German' | French: 'S6 586 Row 59 Spare Message French'
  587 = 'Spare' | German: 'S6 587 Row 59 Spare Message German' | French: 'S6 587 Row 59 Spare Message French'
  588 = 'Spare' | German: 'S6 588 Row 59 Spare Message German' | French: 'S6 588 Row 59 Spare Message French'
  589 = 'Spare' | German: 'S6 589 Row 59 Spare Message German' | French: 'S6 589 Row 59 Spare Message French'
  590 = 'Clamp Cylinder A1 Failed to Advance... Check Q1.0...' | German: 'S6 590 Row 60 Failed To Advance.. Check Qxxx.x German' | French: 'S6 590 Row 60 Failed To Advance.. Check Qxxx.x French'
  591 = 'Clamp Cylinder A1 Failed to Return... Check Q1.1...' | German: 'S6 591 Row 60 Failed To Return.. Check Qxxx.x German' | French: 'S6 591 Row 60 Failed To Return.. Check Qxxx.x French'
  592 = 'Clamp Cylinder A1 Lost Advanced... Check I1.0...' | German: 'S6 592 Row 60 Lost Advance Position... Check Ixxx.x German' | French: 'S6 592 Row 60 Lost Advance Position... Check Ixxx.x French'
  593 = 'Clamp Cylinder A1 Lost Returned... Check I1.1...' | German: 'S6 593 Row 60 Lost Return Position... Check Ixxx.x German' | French: 'S6 593 Row 60 Lost Return Position... Check Ixxx.x French'
  594 = 'Clamp Cylinder A1 Switch Fault... Check I1.0, I1.1...' | German: 'S6 594 Row 60 Switch Fault... Check Ixxx.x / Ixxx.x German' | French: 'S6 594 Row 60 Switch Fault... Check Ixxx.x / Ixxx.x French'
  595 = 'Spare' | German: 'S6 595 Row 60 Spare Message German' | French: 'S6 595 Row 60 Spare Message French'
  596 = 'Spare' | German: 'S6 596 Row 60 Spare Message German' | French: 'S6 596 Row 60 Spare Message French'
  597 = 'Spare' | German: 'S6 597 Row 60 Spare Message German' | French: 'S6 597 Row 60 Spare Message French'
  598 = 'Spare' | German: 'S6 598 Row 60 Spare Message German' | French: 'S6 598 Row 60 Spare Message French'
  599 = 'Spare' | German: 'S6 599 Row 60 Spare Message German' | French: 'S6 599 Row 60 Spare Message French'
  600 = 'Clamp Cylinder A1 Failed to Advance... Check Q1.0...' | German: 'S6 600 Row 61 Failed To Advance.. Check Qxxx.x German' | French: 'S6 600 Row 61 Failed To Advance.. Check Qxxx.x French'
  601 = 'Clamp Cylinder A1 Failed to Return... Check Q1.1...' | German: 'S6 601 Row 61 Failed To Return.. Check Qxxx.x German' | French: 'S6 601 Row 61 Failed To Return.. Check Qxxx.x French'
  602 = 'Clamp Cylinder A1 Lost Advanced... Check I1.0...' | German: 'S6 602 Row 61 Lost Advance Position... Check Ixxx.x German' | French: 'S6 602 Row 61 Lost Advance Position... Check Ixxx.x French'
  603 = 'Clamp Cylinder A1 Lost Returned... Check I1.1...' | German: 'S6 603 Row 61 Lost Return Position... Check Ixxx.x German' | French: 'S6 603 Row 61 Lost Return Position... Check Ixxx.x French'
  604 = 'Clamp Cylinder A1 Switch Fault... Check I1.0, I1.1...' | German: 'S6 604 Row 61 Switch Fault... Check Ixxx.x / Ixxx.x German' | French: 'S6 604 Row 61 Switch Fault... Check Ixxx.x / Ixxx.x French'
  605 = 'Spare' | German: 'S6 605 Row 61 Spare Message German' | French: 'S6 605 Row 61 Spare Message French'
  606 = 'Spare' | German: 'S6 606 Row 61 Spare Message German' | French: 'S6 606 Row 61 Spare Message French'
  607 = 'Spare' | German: 'S6 607 Row 61 Spare Message German' | French: 'S6 607 Row 61 Spare Message French'
  608 = 'Spare' | German: 'S6 608 Row 61 Spare Message German' | French: 'S6 608 Row 61 Spare Message French'
  609 = 'Spare' | German: 'S6 609 Row 61 Spare Message German' | French: 'S6 609 Row 61 Spare Message French'
  610 = 'Clamp Cylinder A1 Failed to Advance... Check Q1.0...' | German: 'S6 610 Row 62 Failed To Advance.. Check Qxxx.x German' | French: 'S6 610 Row 62 Failed To Advance.. Check Qxxx.x French'
  611 = 'Clamp Cylinder A1 Failed to Return... Check Q1.1...' | German: 'S6 611 Row 62 Failed To Return.. Check Qxxx.x German' | French: 'S6 611 Row 62 Failed To Return.. Check Qxxx.x French'
  612 = 'Clamp Cylinder A1 Lost Advanced... Check I1.0...' | German: 'S6 612 Row 62 Lost Advance Position... Check Ixxx.x German' | French: 'S6 612 Row 62 Lost Advance Position... Check Ixxx.x French'
  613 = 'Clamp Cylinder A1 Lost Returned... Check I1.1...' | German: 'S6 613 Row 62 Lost Return Position... Check Ixxx.x German' | French: 'S6 613 Row 62 Lost Return Position... Check Ixxx.x French'
  614 = 'Clamp Cylinder A1 Switch Fault... Check I1.0, I1.1...' | German: 'S6 614 Row 62 Switch Fault... Check Ixxx.x / Ixxx.x German' | French: 'S6 614 Row 62 Switch Fault... Check Ixxx.x / Ixxx.x French'
  615 = 'Spare' | German: 'S6 615 Row 62 Spare Message German' | French: 'S6 615 Row 62 Spare Message French'
  616 = 'Spare' | German: 'S6 616 Row 62 Spare Message German' | French: 'S6 616 Row 62 Spare Message French'
  617 = 'Spare' | German: 'S6 617 Row 62 Spare Message German' | French: 'S6 617 Row 62 Spare Message French'
  618 = 'Spare' | German: 'S6 618 Row 62 Spare Message German' | French: 'S6 618 Row 62 Spare Message French'
  619 = 'Spare' | German: 'S6 619 Row 62 Spare Message German' | French: 'S6 619 Row 62 Spare Message French'
  620 = 'Clamp Cylinder A1 Failed to Advance... Check Q1.0...' | German: 'S6 620 Row 63 Failed To Advance.. Check Qxxx.x German' | French: 'S6 620 Row 63 Failed To Advance.. Check Qxxx.x French'
  621 = 'Clamp Cylinder A1 Failed to Return... Check Q1.1...' | German: 'S6 621 Row 63 Failed To Return.. Check Qxxx.x German' | French: 'S6 621 Row 63 Failed To Return.. Check Qxxx.x French'
  622 = 'Clamp Cylinder A1 Lost Advanced... Check I1.0...' | German: 'S6 622 Row 63 Lost Advance Position... Check Ixxx.x German' | French: 'S6 622 Row 63 Lost Advance Position... Check Ixxx.x French'
  623 = 'Clamp Cylinder A1 Lost Returned... Check I1.1...' | German: 'S6 623 Row 63 Lost Return Position... Check Ixxx.x German' | French: 'S6 623 Row 63 Lost Return Position... Check Ixxx.x French'
  624 = 'Clamp Cylinder A1 Switch Fault... Check I1.0, I1.1...' | German: 'S6 624 Row 63 Switch Fault... Check Ixxx.x / Ixxx.x German' | French: 'S6 624 Row 63 Switch Fault... Check Ixxx.x / Ixxx.x French'
  625 = 'Spare' | German: 'S6 625 Row 63 Spare Message German' | French: 'S6 625 Row 63 Spare Message French'
  626 = 'Spare' | German: 'S6 626 Row 63 Spare Message German' | French: 'S6 626 Row 63 Spare Message French'
  627 = 'Spare' | German: 'S6 627 Row 63 Spare Message German' | French: 'S6 627 Row 63 Spare Message French'
  628 = 'Spare' | German: 'S6 628 Row 63 Spare Message German' | French: 'S6 628 Row 63 Spare Message French'
  629 = 'Spare' | German: 'S6 629 Row 63 Spare Message German' | French: 'S6 629 Row 63 Spare Message French'
  630 = 'Clamp Cylinder A1 Failed to Advance... Check Q1.0...' | German: 'S6 630 Row 64 Failed To Advance.. Check Qxxx.x German' | French: 'S6 630 Row 64 Failed To Advance.. Check Qxxx.x French'
  631 = 'Clamp Cylinder A1 Failed to Return... Check Q1.1...' | German: 'S6 631 Row 64 Failed To Return.. Check Qxxx.x German' | French: 'S6 631 Row 64 Failed To Return.. Check Qxxx.x French'
  632 = 'Clamp Cylinder A1 Lost Advanced... Check I1.0...' | German: 'S6 632 Row 64 Lost Advance Position... Check Ixxx.x German' | French: 'S6 632 Row 64 Lost Advance Position... Check Ixxx.x French'
  633 = 'Clamp Cylinder A1 Lost Returned... Check I1.1...' | German: 'S6 633 Row 64 Lost Return Position... Check Ixxx.x German' | French: 'S6 633 Row 64 Lost Return Position... Check Ixxx.x French'
  634 = 'Clamp Cylinder A1 Switch Fault... Check I1.0, I1.1...' | German: 'S6 634 Row 64 Switch Fault... Check Ixxx.x / Ixxx.x German' | French: 'S6 634 Row 64 Switch Fault... Check Ixxx.x / Ixxx.x French'
  635 = 'Spare' | German: 'S6 635 Row 64 Spare Message German' | French: 'S6 635 Row 64 Spare Message French'
  636 = 'Spare' | German: 'S6 636 Row 64 Spare Message German' | French: 'S6 636 Row 64 Spare Message French'
  637 = 'Spare' | German: 'S6 637 Row 64 Spare Message German' | French: 'S6 637 Row 64 Spare Message French'
  638 = 'Spare' | German: 'S6 638 Row 64 Spare Message German' | French: 'S6 638 Row 64 Spare Message French'
  639 = 'Spare' | German: 'S6 639 Row 64 Spare Message German' | French: 'S6 639 Row 64 Spare Message French'
  640 = 'Clamp Cylinder A1 Failed to Advance... Check Q1.0...' | German: 'S6 640 Row 65 Failed To Advance.. Check Qxxx.x German' | French: 'S6 640 Row 65 Failed To Advance.. Check Qxxx.x French'
  641 = 'Clamp Cylinder A1 Failed to Return... Check Q1.1...' | German: 'S6 641 Row 65 Failed To Return.. Check Qxxx.x German' | French: 'S6 641 Row 65 Failed To Return.. Check Qxxx.x French'
  642 = 'Clamp Cylinder A1 Lost Advanced... Check I1.0...' | German: 'S6 642 Row 65 Lost Advance Position... Check Ixxx.x German' | French: 'S6 642 Row 65 Lost Advance Position... Check Ixxx.x French'
  643 = 'Clamp Cylinder A1 Lost Returned... Check I1.1...' | German: 'S6 643 Row 65 Lost Return Position... Check Ixxx.x German' | French: 'S6 643 Row 65 Lost Return Position... Check Ixxx.x French'
  644 = 'Clamp Cylinder A1 Switch Fault... Check I1.0, I1.1...' | German: 'S6 644 Row 65 Switch Fault... Check Ixxx.x / Ixxx.x German' | French: 'S6 644 Row 65 Switch Fault... Check Ixxx.x / Ixxx.x French'
  645 = 'Spare' | German: 'S6 645 Row 65 Spare Message German' | French: 'S6 645 Row 65 Spare Message French'
  646 = 'Spare' | German: 'S6 646 Row 65 Spare Message German' | French: 'S6 646 Row 65 Spare Message French'
  647 = 'Spare' | German: 'S6 647 Row 65 Spare Message German' | French: 'S6 647 Row 65 Spare Message French'
  648 = 'Spare' | German: 'S6 648 Row 65 Spare Message German' | French: 'S6 648 Row 65 Spare Message French'
  649 = 'Spare' | German: 'S6 649 Row 65 Spare Message German' | French: 'S6 649 Row 65 Spare Message French'
